LIN {X 0,Y 608.078,Z 640.045,A -85,B 0,C 180,E1 25976.717,E2 25976.717} C_VEL
LIN {X 0,Y 611.182,Z 594.743,A -85,B 0,C 180,E1 25973.511,E2 25973.511} C_VEL
LIN {X 0,Y 614.526,Z 550.793,A -85,B 0,C 180,E1 25970.32,E2 25970.32} C_VEL
LIN {X 0,Y 606.763,Z 531.048,A -85,B 0,C 180,E1 25968.076,E2 25968.076} C_VEL
LIN {X 0,Y 599.121,Z 513.107,A -85,B 0,C 180,E1 25965.86,E2 25965.86} C_VEL
LIN {X 0,Y 593.255,Z 499.729,A -85,B 0,C 180,E1 25964.077,E2 25964.077} C_VEL
LIN {X 0,Y 593.169,Z 499.296,A -85,B 0,C 180,E1 25963.406,E2 25963.406} C_VEL
LIN {X 0,Y 593.199,Z 499.34,A -85,B 0,C 180,E1 25960.21,E2 25960.21} C_VEL
LIN {X 0,Y 593.16,Z 499.3,A -85,B 0,C 180,E1 25956.966,E2 25956.966} C_VEL
LIN {X 0,Y 593.195,Z 499.329,A -85,B 0,C 180,E1 25953.797,E2 25953.797} C_VEL
LIN {X 0,Y 593.163,Z 499.335,A -85,B 0,C 180,E1 25950.603,E2 25950.603} C_VEL
LIN {X 0,Y 593.197,Z 499.328,A -85,B 0,C 180,E1 25947.398,E2 25947.398} C_VEL
LIN {X 0,Y 593.171,Z 499.341,A -85,B 0,C 180,E1 25944.181,E2 25944.181} C_VEL
LIN {X 0,Y 593.176,Z 499.338,A -85,B 0,C 180,E1 25940.835,E2 25940.835} C_VEL
LIN {X 0,Y 593.193,Z 499.334,A -85,B 0,C 180,E1 25937.663,E2 25937.663} C_VEL
LIN {X 0,Y 593.16,Z 499.324,A -85,B 0,C 180,E1 25934.447,E2 25934.447} C_VEL
LIN {X 0,Y 593.196,Z 499.326,A -85,B 0,C 180,E1 25931.276,E2 25931.276} C_VEL
LIN {X 0,Y 593.156,Z 499.342,A -85,B 0,C 180,E1 25928.043,E2 25928.043} C_VEL
LIN {X 0,Y 593.195,Z 499.331,A -85,B 0,C 180,E1 25924.835,E2 25924.835} C_VEL
LIN {X 0,Y 593.153,Z 499.332,A -85,B 0,C 180,E1 25921.739,E2 25921.739} C_VEL
LIN {X 0,Y 593.197,Z 499.336,A -85,B 0,C 180,E1 25918.551,E2 25918.551} C_VEL
LIN {X 0,Y 593.16,Z 499.332,A -85,B 0,C 180,E1 25915.359,E2 25915.359} C_VEL
LIN {X 0,Y 593.171,Z 499.319,A -85,B 0,C 180,E1 25912.055,E2 25912.055} C_VEL
LIN {X 0,Y 593.18,Z 499.34,A -85,B 0,C 180,E1 25908.921,E2 25908.921} C_VEL
LIN {X 0,Y 593.156,Z 499.34,A -85,B 0,C 180,E1 25905.653,E2 25905.653} C_VEL
LIN {X 0,Y 593.194,Z 499.326,A -85,B 0,C 180,E1 25902.54,E2 25902.54} C_VEL
LIN {X 0,Y 593.149,Z 499.33,A -85,B 0,C 180,E1 25899.317,E2 25899.317} C_VEL
LIN {X 0,Y 593.201,Z 499.331,A -85,B 0,C 180,E1 25896.24,E2 25896.24} C_VEL
LIN {X 0,Y 593.148,Z 499.344,A -85,B 0,C 180,E1 25893.034,E2 25893.034} C_VEL
LIN {X 0,Y 593.204,Z 499.341,A -85,B 0,C 180,E1 25889.959,E2 25889.959} C_VEL
LIN {X 0,Y 593.14,Z 499.291,A -85,B 0,C 180,E1 25886.779,E2 25886.779} C_VEL
LIN {X 0,Y 593.196,Z 499.341,A -85,B 0,C 180,E1 25883.606,E2 25883.606} C_VEL
LIN {X 0,Y 593.14,Z 499.296,A -85,B 0,C 180,E1 25880.538,E2 25880.538} C_VEL
LIN {X 0,Y 593.188,Z 499.306,A -85,B 0,C 180,E1 25877.342,E2 25877.342} C_VEL
LIN {X 0,Y 593.176,Z 499.54,A -85,B 0,C 180,E1 25876.313,E2 25876.313} C_VEL
LIN {X 0,Y 594.452,Z 502.746,A -85,B 0,C 180,E1 25875.864,E2 25875.864} C_VEL
LIN {X 0,Y 602.44,Z 520.278,A -85,B 0,C 180,E1 25873.643,E2 25873.643} C_VEL
LIN {X 0,Y 609.643,Z 537.266,A -85,B 0,C 180,E1 25871.662,E2 25871.662} C_VEL
LIN {X 0,Y 610.94,Z 539.957,A -85,B 0,C 180,E1 25871.41,E2 25871.41} C_VEL
LIN {X 0,Y 619.493,Z 554.552,A -85,B 0,C 180,E1 25870.572,E2 25870.572} C_VEL
LIN {X 0,Y 620.819,Z 562.667,A -85,B 0,C 180,E1 25870.357,E2 25870.357} C_VEL
LIN {X 0,Y 615.586,Z 815.185,A -85,B 0,C 180,E1 25866.946,E2 25866.946} C_VEL
LIN {X 0,Y 613.51,Z 921.471,A -85,B 0,C 180,E1 25865.506,E2 25865.506} C_VEL
LIN {X 0,Y 612.502,Z 946.347,A -85,B 0,C 180,E1 25865.008,E2 25865.008} C_VEL
LIN {X 0,Y 611.446,Z 967.057,A -85,B 0,C 180,E1 25864.465,E2 25864.465} C_VEL
LIN {X 0,Y 609.921,Z 992.831,A -85,B 0,C 180,E1 25863.612,E2 25863.612} C_VEL
LIN {X 0,Y 608.442,Z 1014.751,A -85,B 0,C 180,E1 25862.728,E2 25862.728} C_VEL
LIN {X 0,Y 606.737,Z 1038.002,A -85,B 0,C 180,E1 25861.604,E2 25861.604} C_VEL
LIN {X 0,Y 605.201,Z 1057.039,A -85,B 0,C 180,E1 25860.532,E2 25860.532} C_VEL
LIN {X 0,Y 603.232,Z 1079.697,A -85,B 0,C 180,E1 25859.055,E2 25859.055} C_VEL
LIN {X 0,Y 601.654,Z 1097.29,A -85,B 0,C 180,E1 25857.731,E2 25857.731} C_VEL
LIN {X 0,Y 599.985,Z 1115.676,A -85,B 0,C 180,E1 25856.154,E2 25856.154} C_VEL
LIN {X 0,Y 598.433,Z 1131.856,A -85,B 0,C 180,E1 25854.555,E2 25854.555} C_VEL
LIN {X 0,Y 596.98,Z 1147.996,A -85,B 0,C 180,E1 25852.761,E2 25852.761} C_VEL
LIN {X 0,Y 595.66,Z 1162.851,A -85,B 0,C 180,E1 25850.846,E2 25850.846} C_VEL
LIN {X 0,Y 594.748,Z 1173.87,A -85,B 0,C 180,E1 25849.239,E2 25849.239} C_VEL
LIN {X 0,Y 593.77,Z 1186.22,A -85,B 0,C 180,E1 25847.139,E2 25847.139} C_VEL
LIN {X 0,Y 593.053,Z 1196.639,A -85,B 0,C 180,E1 25845.048,E2 25845.048} C_VEL
LIN {X 0,Y 592.568,Z 1205.584,A -85,B 0,C 180,E1 25842.968,E2 25842.968} C_VEL
LIN {X 0,Y 592.211,Z 1213.908,A -85,B 0,C 180,E1 25840.605,E2 25840.605} C_VEL
LIN {X 0,Y 592.044,Z 1219.746,A -85,B 0,C 180,E1 25838.547,E2 25838.547} C_VEL
LIN {X 0,Y 591.951,Z 1225.015,A -85,B 0,C 180,E1 25836.109,E2 25836.109} C_VEL
LIN {X 0,Y 591.917,Z 1228.122,A -85,B 0,C 180,E1 25833.971,E2 25833.971} C_VEL
LIN {X 0,Y 591.899,Z 1230.037,A -85,B 0,C 180,E1 25831.742,E2 25831.742} C_VEL
LIN {X 0,Y 591.884,Z 1230.371,A -85,B 0,C 180,E1 25829.419,E2 25829.419} C_VEL
LIN {X 0,Y 591.892,Z 1229.426,A -85,B 0,C 180,E1 25827.386,E2 25827.386} C_VEL
LIN {X 0,Y 591.906,Z 1226.929,A -85,B 0,C 180,E1 25825.058,E2 25825.058} C_VEL
LIN {X 0,Y 591.973,Z 1223.102,A -85,B 0,C 180,E1 25822.917,E2 25822.917} C_VEL
LIN {X 0,Y 592.071,Z 1218.22,A -85,B 0,C 180,E1 25820.866,E2 25820.866} C_VEL
LIN {X 0,Y 592.321,Z 1210.66,A -85,B 0,C 180,E1 25818.412,E2 25818.412} C_VEL
LIN {X 0,Y 592.677,Z 1203.153,A -85,B 0,C 180,E1 25816.438,E2 25816.438} C_VEL
LIN {X 0,Y 593.283,Z 1193.273,A -85,B 0,C 180,E1 25814.226,E2 25814.226} C_VEL
LIN {X 0,Y 594.113,Z 1181.687,A -85,B 0,C 180,E1 25812.063,E2 25812.063} C_VEL
LIN {X 0,Y 595.01,Z 1170.617,A -85,B 0,C 180,E1 25810.259,E2 25810.259} C_VEL
LIN {X 0,Y 596.311,Z 1155.263,A -85,B 0,C 180,E1 25808.146,E2 25808.146} C_VEL
LIN {X 0,Y 597.61,Z 1140.965,A -85,B 0,C 180,E1 25806.43,E2 25806.43} C_VEL
LIN {X 0,Y 599.308,Z 1122.566,A -85,B 0,C 180,E1 25804.504,E2 25804.504} C_VEL
LIN {X 0,Y 600.868,Z 1105.911,A -85,B 0,C 180,E1 25802.982,E2 25802.982} C_VEL
LIN {X 0,Y 602.8,Z 1084.729,A -85,B 0,C 180,E1 25801.308,E2 25801.308} C_VEL
LIN {X 0,Y 604.418,Z 1066.075,A -85,B 0,C 180,E1 25800.028,E2 25800.028} C_VEL
LIN {X 0,Y 606.349,Z 1042.88,A -85,B 0,C 180,E1 25798.656,E2 25798.656} C_VEL
LIN {X 0,Y 607.897,Z 1022.873,A -85,B 0,C 180,E1 25797.644,E2 25797.644} C_VEL
LIN {X 0,Y 609.578,Z 998.087,A -85,B 0,C 180,E1 25796.586,E2 25796.586} C_VEL
LIN {X 0,Y 610.944,Z 975.646,A -85,B 0,C 180,E1 25795.794,E2 25795.794} C_VEL
LIN {X 0,Y 612.299,Z 950.422,A -85,B 0,C 180,E1 25795.088,E2 25795.088} C_VEL
LIN {X 0,Y 613.253,Z 928.821,A -85,B 0,C 180,E1 25794.626,E2 25794.626} C_VEL
LIN {X 0,Y 614.11,Z 895.917,A -85,B 0,C 180,E1 25794.131,E2 25794.131} C_VEL
LIN {X 0,Y 618.886,Z 652.893,A -85,B 0,C 180,E1 25790.86,E2 25790.86} C_VEL
LIN {X 0,Y 620.673,Z 560.775,A -85,B 0,C 180,E1 25789.605,E2 25789.605} C_VEL
LIN {X 0,Y 619.085,Z 553.518,A -85,B 0,C 180,E1 25789.385,E2 25789.385} C_VEL
LIN {X 0,Y 610.437,Z 539.117,A -85,B 0,C 180,E1 25788.537,E2 25788.537} C_VEL
LIN {X 0,Y 603.016,Z 521.573,A -85,B 0,C 180,E1 25786.519,E2 25786.519} C_VEL
LIN {X 0,Y 594.856,Z 503.322,A -85,B 0,C 180,E1 25784.233,E2 25784.233} C_VEL
LIN {X 0,Y 593.189,Z 499.611,A -85,B 0,C 180,E1 25783.718,E2 25783.718} C_VEL
LIN {X 0,Y 593.195,Z 499.309,A -85,B 0,C 180,E1 25782.526,E2 25782.526} C_VEL
LIN {X 0,Y 593.141,Z 499.295,A -85,B 0,C 180,E1 25779.46,E2 25779.46} C_VEL
LIN {X 0,Y 593.2,Z 499.341,A -85,B 0,C 180,E1 25776.324,E2 25776.324} C_VEL
LIN {X 0,Y 593.142,Z 499.291,A -85,B 0,C 180,E1 25773.106,E2 25773.106} C_VEL
LIN {X 0,Y 593.203,Z 499.342,A -85,B 0,C 180,E1 25769.929,E2 25769.929} C_VEL
LIN {X 0,Y 593.152,Z 499.343,A -85,B 0,C 180,E1 25766.858,E2 25766.858} C_VEL
LIN {X 0,Y 593.199,Z 499.333,A -85,B 0,C 180,E1 25763.651,E2 25763.651} C_VEL
LIN {X 0,Y 593.156,Z 499.331,A -85,B 0,C 180,E1 25760.526,E2 25760.526} C_VEL
LIN {X 0,Y 593.18,Z 499.327,A -85,B 0,C 180,E1 25757.258,E2 25757.258} C_VEL
LIN {X 0,Y 593.171,Z 499.339,A -85,B 0,C 180,E1 25754.148,E2 25754.148} C_VEL
LIN {X 0,Y 593.163,Z 499.344,A -85,B 0,C 180,E1 25750.784,E2 25750.784} C_VEL
LIN {X 0,Y 593.198,Z 499.317,A -85,B 0,C 180,E1 25747.652,E2 25747.652} C_VEL
LIN {X 0,Y 593.157,Z 499.329,A -85,B 0,C 180,E1 25744.447,E2 25744.447} C_VEL
LIN {X 0,Y 593.197,Z 499.337,A -85,B 0,C 180,E1 25741.256,E2 25741.256} C_VEL
LIN {X 0,Y 593.157,Z 499.334,A -85,B 0,C 180,E1 25738.068,E2 25738.068} C_VEL
LIN {X 0,Y 593.195,Z 499.327,A -85,B 0,C 180,E1 25734.875,E2 25734.875} C_VEL
LIN {X 0,Y 593.166,Z 499.339,A -85,B 0,C 180,E1 25731.675,E2 25731.675} C_VEL
LIN {X 0,Y 593.183,Z 499.335,A -85,B 0,C 180,E1 25728.328,E2 25728.328} C_VEL
LIN {X 0,Y 593.199,Z 499.319,A -85,B 0,C 180,E1 25725.055,E2 25725.055} C_VEL
LIN {X 0,Y 593.166,Z 499.33,A -85,B 0,C 180,E1 25721.829,E2 25721.829} C_VEL
LIN {X 0,Y 593.196,Z 499.339,A -85,B 0,C 180,E1 25718.648,E2 25718.648} C_VEL
LIN {X 0,Y 593.166,Z 499.343,A -85,B 0,C 180,E1 25715.501,E2 25715.501} C_VEL
LIN {X 0,Y 593.194,Z 499.331,A -85,B 0,C 180,E1 25712.275,E2 25712.275} C_VEL
LIN {X 0,Y 593.169,Z 499.337,A -85,B 0,C 180,E1 25709.09,E2 25709.09} C_VEL
LIN {X 0,Y 593.194,Z 499.332,A -85,B 0,C 180,E1 25705.853,E2 25705.853} C_VEL
LIN {X 0,Y 593.178,Z 499.293,A -85,B 0,C 180,E1 25702.639,E2 25702.639} C_VEL
LIN {X 0,Y 593.179,Z 499.342,A -85,B 0,C 180,E1 25699.281,E2 25699.281} C_VEL
LIN {X 0,Y 593.198,Z 499.367,A -85,B 0,C 180,E1 25696.015,E2 25696.015} C_VEL
LIN {X 0,Y 593.297,Z 499.956,A -85,B 0,C 180,E1 25695.79,E2 25695.79} C_VEL
LIN {X 0,Y 601.72,Z 518.947,A -85,B 0,C 180,E1 25693.295,E2 25693.295} C_VEL
LIN {X 0,Y 610.485,Z 540.277,A -85,B 0,C 180,E1 25690.754,E2 25690.754} C_VEL
LIN {X 0,Y 614.495,Z 551.086,A -85,B 0,C 180,E1 25689.564,E2 25689.564} C_VEL
LIN {X 0,Y 611.039,Z 596.556,A -85,B 0,C 180,E1 25686.266,E2 25686.266} C_VEL
LIN {X 0,Y 608.667,Z 630.364,A -85,B 0,C 180,E1 25683.868,E2 25683.868} C_VEL
LIN {X 0,Y 607.998,Z 636.114,A -85,B 0,C 180,E1 25683.565,E2 25683.565} C_VEL
LIN {X 0,Y 606.57,Z 644.568,A -85,B 0,C 180,E1 25683.334,E2 25683.334} C_VEL
LIN {X 0,Y 605.188,Z 656.769,A -85,B 0,C 180,E1 25683.155,E2 25683.155} C_VEL
LIN {X 0,Y 605.693,Z 664.458,A -85,B 0,C 180,E1 25683.005,E2 25683.005} C_VEL
LIN {X 0,Y 608.402,Z 681.191,A -85,B 0,C 180,E1 25682.592,E2 25682.592} C_VEL
LIN {X 0,Y 604.985,Z 954.452,A -85,B 0,C 180,E1 25679.305,E2 25679.305} C_VEL
LIN {X 0,Y 604.101,Z 976.225,A -85,B 0,C 180,E1 25678.892,E2 25678.892} C_VEL
LIN {X 0,Y 602.959,Z 997.031,A -85,B 0,C 180,E1 25678.338,E2 25678.338} C_VEL
LIN {X 0,Y 601.467,Z 1017.095,A -85,B 0,C 180,E1 25677.632,E2 25677.632} C_VEL
LIN {X 0,Y 599.717,Z 1037.712,A -85,B 0,C 180,E1 25676.726,E2 25676.726} C_VEL
LIN {X 0,Y 597.899,Z 1056.39,A -85,B 0,C 180,E1 25675.73,E2 25675.73} C_VEL
LIN {X 0,Y 595.886,Z 1074.87,A -85,B 0,C 180,E1 25674.543,E2 25674.543} C_VEL
LIN {X 0,Y 593.817,Z 1093.059,A -85,B 0,C 180,E1 25673.164,E2 25673.164} C_VEL
LIN {X 0,Y 591.871,Z 1109.557,A -85,B 0,C 180,E1 25671.696,E2 25671.696} C_VEL
LIN {X 0,Y 590.071,Z 1124.599,A -85,B 0,C 180,E1 25670.119,E2 25670.119} C_VEL
LIN {X 0,Y 588.473,Z 1138.59,A -85,B 0,C 180,E1 25668.423,E2 25668.423} C_VEL
LIN {X 0,Y 587.093,Z 1151.213,A -85,B 0,C 180,E1 25666.625,E2 25666.625} C_VEL
LIN {X 0,Y 585.924,Z 1163.106,A -85,B 0,C 180,E1 25664.625,E2 25664.625} C_VEL
LIN {X 0,Y 585.071,Z 1173.557,A -85,B 0,C 180,E1 25662.535,E2 25662.535} C_VEL
LIN {X 0,Y 584.502,Z 1182.555,A -85,B 0,C 180,E1 25660.347,E2 25660.347} C_VEL
LIN {X 0,Y 584.169,Z 1189.59,A -85,B 0,C 180,E1 25658.167,E2 25658.167} C_VEL
LIN {X 0,Y 583.993,Z 1194.928,A -85,B 0,C 180,E1 25655.995,E2 25655.995} C_VEL
LIN {X 0,Y 583.94,Z 1198.661,A -85,B 0,C 180,E1 25653.829,E2 25653.829} C_VEL
LIN {X 0,Y 583.918,Z 1200.67,A -85,B 0,C 180,E1 25651.668,E2 25651.668} C_VEL
LIN {X 0,Y 583.911,Z 1201.109,A -85,B 0,C 180,E1 25649.411,E2 25649.411} C_VEL
LIN {X 0,Y 583.927,Z 1199.973,A -85,B 0,C 180,E1 25647.252,E2 25647.252} C_VEL
LIN {X 0,Y 583.953,Z 1197.131,A -85,B 0,C 180,E1 25645.089,E2 25645.089} C_VEL
LIN {X 0,Y 584.053,Z 1192.685,A -85,B 0,C 180,E1 25642.92,E2 25642.92} C_VEL
LIN {X 0,Y 584.301,Z 1186.601,A -85,B 0,C 180,E1 25640.744,E2 25640.744} C_VEL
LIN {X 0,Y 584.701,Z 1179.023,A -85,B 0,C 180,E1 25638.659,E2 25638.659} C_VEL
LIN {X 0,Y 585.363,Z 1169.714,A -85,B 0,C 180,E1 25636.567,E2 25636.567} C_VEL
LIN {X 0,Y 586.305,Z 1159.134,A -85,B 0,C 180,E1 25634.572,E2 25634.572} C_VEL
LIN {X 0,Y 587.525,Z 1147.139,A -85,B 0,C 180,E1 25632.674,E2 25632.674} C_VEL
LIN {X 0,Y 589.006,Z 1133.769,A -85,B 0,C 180,E1 25630.875,E2 25630.875} C_VEL
LIN {X 0,Y 590.734,Z 1119.091,A -85,B 0,C 180,E1 25629.18,E2 25629.18} C_VEL
LIN {X 0,Y 592.539,Z 1103.888,A -85,B 0,C 180,E1 25627.687,E2 25627.687} C_VEL
LIN {X 0,Y 594.603,Z 1086.209,A -85,B 0,C 180,E1 25626.198,E2 25626.198} C_VEL
LIN {X 0,Y 596.657,Z 1068.291,A -85,B 0,C 180,E1 25624.915,E2 25624.915} C_VEL
LIN {X 0,Y 598.575,Z 1049.526,A -85,B 0,C 180,E1 25623.794,E2 25623.794} C_VEL
LIN {X 0,Y 600.524,Z 1028.723,A -85,B 0,C 180,E1 25622.764,E2 25622.764} C_VEL
LIN {X 0,Y 602.141,Z 1009.074,A -85,B 0,C 180,E1 25621.971,E2 25621.971} C_VEL
LIN {X 0,Y 603.476,Z 987.858,A -85,B 0,C 180,E1 25621.307,E2 25621.307} C_VEL
LIN {X 0,Y 604.607,Z 965.172,A -85,B 0,C 180,E1 25620.787,E2 25620.787} C_VEL
LIN {X 0,Y 605.264,Z 943.024,A -85,B 0,C 180,E1 25620.449,E2 25620.449} C_VEL
LIN {X 0,Y 608.386,Z 679.678,A -85,B 0,C 180,E1 25617.291,E2 25617.291} C_VEL
LIN {X 0,Y 601.204,Z 639.323,A -85,B 0,C 180,E1 25616.223,E2 25616.223} C_VEL
LIN {X 0,Y 604.486,Z 594.03,A -85,B 0,C 180,E1 25612.981,E2 25612.981} C_VEL
LIN {X 0,Y 607.7,Z 554.273,A -85,B 0,C 180,E1 25610.063,E2 25610.063} C_VEL
LIN {X 0,Y 599.505,Z 533.257,A -85,B 0,C 180,E1 25607.635,E2 25607.635} C_VEL
LIN {X 0,Y 591.378,Z 514.462,A -85,B 0,C 180,E1 25605.246,E2 25605.246} C_VEL
LIN {X 0,Y 586.57,Z 503.804,A -85,B 0,C 180,E1 25603.796,E2 25603.796} C_VEL
LIN {X 0,Y 585.256,Z 500.501,A -85,B 0,C 180,E1 25603.299,E2 25603.299} C_VEL
LIN {X 0,Y 585.26,Z 500.329,A -85,B 0,C 180,E1 25600.213,E2 25600.213} C_VEL
LIN {X 0,Y 585.221,Z 500.287,A -85,B 0,C 180,E1 25596.972,E2 25596.972} C_VEL
LIN {X 0,Y 585.256,Z 500.317,A -85,B 0,C 180,E1 25593.846,E2 25593.846} C_VEL
LIN {X 0,Y 585.224,Z 500.323,A -85,B 0,C 180,E1 25590.607,E2 25590.607} C_VEL
LIN {X 0,Y 585.257,Z 500.316,A -85,B 0,C 180,E1 25587.331,E2 25587.331} C_VEL
LIN {X 0,Y 585.237,Z 500.326,A -85,B 0,C 180,E1 25584.101,E2 25584.101} C_VEL
LIN {X 0,Y 585.23,Z 500.328,A -85,B 0,C 180,E1 25580.712,E2 25580.712} C_VEL
LIN {X 0,Y 585.258,Z 500.326,A -85,B 0,C 180,E1 25577.499,E2 25577.499} C_VEL
LIN {X 0,Y 585.217,Z 500.314,A -85,B 0,C 180,E1 25574.243,E2 25574.243} C_VEL
LIN {X 0,Y 585.256,Z 500.31,A -85,B 0,C 180,E1 25571.032,E2 25571.032} C_VEL
LIN {X 0,Y 585.22,Z 500.332,A -85,B 0,C 180,E1 25567.856,E2 25567.856} C_VEL
LIN {X 0,Y 585.251,Z 500.325,A -85,B 0,C 180,E1 25564.606,E2 25564.606} C_VEL
LIN {X 0,Y 585.226,Z 500.316,A -85,B 0,C 180,E1 25561.469,E2 25561.469} C_VEL
LIN {X 0,Y 585.227,Z 500.327,A -85,B 0,C 180,E1 25558.129,E2 25558.129} C_VEL
LIN {X 0,Y 585.255,Z 500.325,A -85,B 0,C 180,E1 25554.903,E2 25554.903} C_VEL
LIN {X 0,Y 585.213,Z 500.31,A -85,B 0,C 180,E1 25551.748,E2 25551.748} C_VEL
LIN {X 0,Y 585.258,Z 500.318,A -85,B 0,C 180,E1 25548.569,E2 25548.569} C_VEL
LIN {X 0,Y 585.209,Z 500.331,A -85,B 0,C 180,E1 25545.352,E2 25545.352} C_VEL
LIN {X 0,Y 585.259,Z 500.319,A -85,B 0,C 180,E1 25542.193,E2 25542.193} C_VEL
LIN {X 0,Y 585.211,Z 500.317,A -85,B 0,C 180,E1 25539.078,E2 25539.078} C_VEL
LIN {X 0,Y 585.257,Z 500.314,A -85,B 0,C 180,E1 25535.9,E2 25535.9} C_VEL
LIN {X 0,Y 585.216,Z 500.333,A -85,B 0,C 180,E1 25532.748,E2 25532.748} C_VEL
LIN {X 0,Y 585.231,Z 500.328,A -85,B 0,C 180,E1 25529.393,E2 25529.393} C_VEL
LIN {X 0,Y 585.228,Z 500.275,A -85,B 0,C 180,E1 25526.27,E2 25526.27} C_VEL
LIN {X 0,Y 585.215,Z 500.326,A -85,B 0,C 180,E1 25523.028,E2 25523.028} C_VEL
LIN {X 0,Y 585.249,Z 500.287,A -85,B 0,C 180,E1 25519.902,E2 25519.902} C_VEL
LIN {X 0,Y 585.256,Z 500.538,A -85,B 0,C 180,E1 25517.032,E2 25517.032} C_VEL
LIN {X 0,Y 586.504,Z 503.773,A -85,B 0,C 180,E1 25516.571,E2 25516.571} C_VEL
LIN {X 0,Y 591.053,Z 513.493,A -85,B 0,C 180,E1 25515.271,E2 25515.271} C_VEL
LIN {X 0,Y 599.255,Z 531.934,A -85,B 0,C 180,E1 25512.974,E2 25512.974} C_VEL
LIN {X 0,Y 602.865,Z 540.477,A -85,B 0,C 180,E1 25512.009,E2 25512.009} C_VEL
LIN {X 0,Y 613.481,Z 558.247,A -85,B 0,C 180,E1 25510.942,E2 25510.942} C_VEL
LIN {X 0,Y 614.388,Z 564.377,A -85,B 0,C 180,E1 25510.783,E2 25510.783} C_VEL
LIN {X 0,Y 608.882,Z 815.259,A -85,B 0,C 180,E1 25507.356,E2 25507.356} C_VEL
LIN {X 0,Y 606.647,Z 921.35,A -85,B 0,C 180,E1 25505.897,E2 25505.897} C_VEL
LIN {X 0,Y 605.592,Z 946.105,A -85,B 0,C 180,E1 25505.396,E2 25505.396} C_VEL
LIN {X 0,Y 604.471,Z 966.709,A -85,B 0,C 180,E1 25504.849,E2 25504.849} C_VEL
LIN {X 0,Y 602.89,Z 991.718,A -85,B 0,C 180,E1 25504.01,E2 25504.01} C_VEL
LIN {X 0,Y 601.315,Z 1013.033,A -85,B 0,C 180,E1 25503.136,E2 25503.136} C_VEL
LIN {X 0,Y 599.374,Z 1037.838,A -85,B 0,C 180,E1 25501.925,E2 25501.925} C_VEL
LIN {X 0,Y 597.77,Z 1056.876,A -85,B 0,C 180,E1 25500.842,E2 25500.842} C_VEL
LIN {X 0,Y 595.71,Z 1079.538,A -85,B 0,C 180,E1 25499.347,E2 25499.347} C_VEL
LIN {X 0,Y 594.056,Z 1097.142,A -85,B 0,C 180,E1 25498.007,E2 25498.007} C_VEL
LIN {X 0,Y 592.271,Z 1116.184,A -85,B 0,C 180,E1 25496.359,E2 25496.359} C_VEL
LIN {X 0,Y 590.707,Z 1132.035,A -85,B 0,C 180,E1 25494.781,E2 25494.781} C_VEL
LIN {X 0,Y 589.192,Z 1148.078,A -85,B 0,C 180,E1 25492.974,E2 25492.974} C_VEL
LIN {X 0,Y 587.812,Z 1162.906,A -85,B 0,C 180,E1 25491.033,E2 25491.033} C_VEL
LIN {X 0,Y 586.788,Z 1174.87,A -85,B 0,C 180,E1 25489.261,E2 25489.261} C_VEL
LIN {X 0,Y 585.746,Z 1188.213,A -85,B 0,C 180,E1 25486.971,E2 25486.971} C_VEL
LIN {X 0,Y 585.12,Z 1197.097,A -85,B 0,C 180,E1 25485.156,E2 25485.156} C_VEL
LIN {X 0,Y 584.563,Z 1206.776,A -85,B 0,C 180,E1 25482.847,E2 25482.847} C_VEL
LIN {X 0,Y 584.21,Z 1214.514,A -85,B 0,C 180,E1 25480.552,E2 25480.552} C_VEL
LIN {X 0,Y 584.047,Z 1220.509,A -85,B 0,C 180,E1 25478.367,E2 25478.367} C_VEL
LIN {X 0,Y 583.947,Z 1225.334,A -85,B 0,C 180,E1 25475.995,E2 25475.995} C_VEL
LIN {X 0,Y 583.916,Z 1228.235,A -85,B 0,C 180,E1 25473.927,E2 25473.927} C_VEL
LIN {X 0,Y 583.897,Z 1230.144,A -85,B 0,C 180,E1 25471.57,E2 25471.57} C_VEL
LIN {X 0,Y 583.885,Z 1230.348,A -85,B 0,C 180,E1 25469.313,E2 25469.313} C_VEL
LIN {X 0,Y 583.891,Z 1229.426,A -85,B 0,C 180,E1 25467.35,E2 25467.35} C_VEL
LIN {X 0,Y 583.905,Z 1226.929,A -85,B 0,C 180,E1 25464.99,E2 25464.99} C_VEL
LIN {X 0,Y 583.971,Z 1223.102,A -85,B 0,C 180,E1 25462.82,E2 25462.82} C_VEL
LIN {X 0,Y 584.091,Z 1218.22,A -85,B 0,C 180,E1 25460.74,E2 25460.74} C_VEL
LIN {X 0,Y 584.364,Z 1210.66,A -85,B 0,C 180,E1 25458.252,E2 25458.252} C_VEL
LIN {X 0,Y 584.746,Z 1203.072,A -85,B 0,C 180,E1 25456.23,E2 25456.23} C_VEL
LIN {X 0,Y 585.416,Z 1192.916,A -85,B 0,C 180,E1 25453.937,E2 25453.937} C_VEL
LIN {X 0,Y 586.215,Z 1181.999,A -85,B 0,C 180,E1 25451.915,E2 25451.915} C_VEL
LIN {X 0,Y 587.201,Z 1170.018,A -85,B 0,C 180,E1 25449.986,E2 25449.986} C_VEL
LIN {X 0,Y 588.494,Z 1155.34,A -85,B 0,C 180,E1 25447.946,E2 25447.946} C_VEL
LIN {X 0,Y 589.854,Z 1141.031,A -85,B 0,C 180,E1 25446.207,E2 25446.207} C_VEL
LIN {X 0,Y 591.607,Z 1122.737,A -85,B 0,C 180,E1 25444.269,E2 25444.269} C_VEL
LIN {X 0,Y 593.247,Z 1105.809,A -85,B 0,C 180,E1 25442.714,E2 25442.714} C_VEL
LIN {X 0,Y 595.263,Z 1084.514,A -85,B 0,C 180,E1 25441.014,E2 25441.014} C_VEL
LIN {X 0,Y 596.993,Z 1065.429,A -85,B 0,C 180,E1 25439.693,E2 25439.693} C_VEL
LIN {X 0,Y 598.985,Z 1042.62,A -85,B 0,C 180,E1 25438.333,E2 25438.333} C_VEL
LIN {X 0,Y 600.704,Z 1021.482,A -85,B 0,C 180,E1 25437.251,E2 25437.251} C_VEL
LIN {X 0,Y 602.446,Z 997.731,A -85,B 0,C 180,E1 25436.221,E2 25436.221} C_VEL
LIN {X 0,Y 603.859,Z 976.413,A -85,B 0,C 180,E1 25435.452,E2 25435.452} C_VEL
LIN {X 0,Y 605.34,Z 950.895,A -85,B 0,C 180,E1 25434.719,E2 25434.719} C_VEL
LIN {X 0,Y 606.335,Z 929.724,A -85,B 0,C 180,E1 25434.256,E2 25434.256} C_VEL
LIN {X 0,Y 607.218,Z 899.395,A -85,B 0,C 180,E1 25433.784,E2 25433.784} C_VEL
LIN {X 0,Y 612.363,Z 653.966,A -85,B 0,C 180,E1 25430.437,E2 25430.437} C_VEL
LIN {X 0,Y 614.25,Z 562.382,A -85,B 0,C 180,E1 25429.177,E2 25429.177} C_VEL
LIN {X 0,Y 613.083,Z 557.386,A -85,B 0,C 180,E1 25429.018,E2 25429.018} C_VEL
LIN {X 0,Y 602.567,Z 539.941,A -85,B 0,C 180,E1 25427.952,E2 25427.952} C_VEL
LIN {X 0,Y 594.327,Z 520.546,A -85,B 0,C 180,E1 25425.645,E2 25425.645} C_VEL
LIN {X 0,Y 587.957,Z 506.912,A -85,B 0,C 180,E1 25423.86,E2 25423.86} C_VEL
LIN {X 0,Y 585.275,Z 500.681,A -85,B 0,C 180,E1 25423.015,E2 25423.015} C_VEL
LIN {X 0,Y 585.259,Z 500.303,A -85,B 0,C 180,E1 25422.291,E2 25422.291} C_VEL
LIN {X 0,Y 585.201,Z 500.28,A -85,B 0,C 180,E1 25419.212,E2 25419.212} C_VEL
LIN {X 0,Y 585.253,Z 500.33,A -85,B 0,C 180,E1 25415.995,E2 25415.995} C_VEL
LIN {X 0,Y 585.215,Z 500.278,A -85,B 0,C 180,E1 25412.794,E2 25412.794} C_VEL
LIN {X 0,Y 585.227,Z 500.326,A -85,B 0,C 180,E1 25409.476,E2 25409.476} C_VEL
LIN {X 0,Y 585.242,Z 500.329,A -85,B 0,C 180,E1 25406.373,E2 25406.373} C_VEL
LIN {X 0,Y 585.219,Z 500.334,A -85,B 0,C 180,E1 25403.14,E2 25403.14} C_VEL
LIN {X 0,Y 585.257,Z 500.318,A -85,B 0,C 180,E1 25399.98,E2 25399.98} C_VEL
LIN {X 0,Y 585.214,Z 500.317,A -85,B 0,C 180,E1 25396.783,E2 25396.783} C_VEL
LIN {X 0,Y 585.262,Z 500.321,A -85,B 0,C 180,E1 25393.637,E2 25393.637} C_VEL
LIN {X 0,Y 585.216,Z 500.33,A -85,B 0,C 180,E1 25390.434,E2 25390.434} C_VEL
LIN {X 0,Y 585.261,Z 500.312,A -85,B 0,C 180,E1 25387.164,E2 25387.164} C_VEL
LIN {X 0,Y 585.223,Z 500.314,A -85,B 0,C 180,E1 25384.017,E2 25384.017} C_VEL
LIN {X 0,Y 585.243,Z 500.327,A -85,B 0,C 180,E1 25380.685,E2 25380.685} C_VEL
LIN {X 0,Y 585.25,Z 500.321,A -85,B 0,C 180,E1 25377.454,E2 25377.454} C_VEL
LIN {X 0,Y 585.224,Z 500.314,A -85,B 0,C 180,E1 25374.214,E2 25374.214} C_VEL
LIN {X 0,Y 585.259,Z 500.327,A -85,B 0,C 180,E1 25371.056,E2 25371.056} C_VEL
LIN {X 0,Y 585.223,Z 500.332,A -85,B 0,C 180,E1 25367.869,E2 25367.869} C_VEL
LIN {X 0,Y 585.255,Z 500.311,A -85,B 0,C 180,E1 25364.644,E2 25364.644} C_VEL
LIN {X 0,Y 585.225,Z 500.316,A -85,B 0,C 180,E1 25361.47,E2 25361.47} C_VEL
LIN {X 0,Y 585.258,Z 500.322,A -85,B 0,C 180,E1 25358.133,E2 25358.133} C_VEL
LIN {X 0,Y 585.253,Z 500.327,A -85,B 0,C 180,E1 25354.823,E2 25354.823} C_VEL
LIN {X 0,Y 585.232,Z 500.333,A -85,B 0,C 180,E1 25351.531,E2 25351.531} C_VEL
LIN {X 0,Y 585.258,Z 500.327,A -85,B 0,C 180,E1 25348.365,E2 25348.365} C_VEL
LIN {X 0,Y 585.232,Z 500.333,A -85,B 0,C 180,E1 25345.085,E2 25345.085} C_VEL
LIN {X 0,Y 585.249,Z 500.276,A -85,B 0,C 180,E1 25341.795,E2 25341.795} C_VEL
LIN {X 0,Y 585.237,Z 500.306,A -85,B 0,C 180,E1 25338.592,E2 25338.592} C_VEL
LIN {X 0,Y 585.274,Z 500.55,A -85,B 0,C 180,E1 25336.579,E2 25336.579} C_VEL
LIN {X 0,Y 588.491,Z 507.938,A -85,B 0,C 180,E1 25335.527,E2 25335.527} C_VEL
LIN {X 0,Y 595.828,Z 524.591,A -85,B 0,C 180,E1 25333.341,E2 25333.341} C_VEL
LIN {X 0,Y 604.237,Z 545.17,A -85,B 0,C 180,E1 25330.866,E2 25330.866} C_VEL
LIN {X 0,Y 607.676,Z 554.478,A -85,B 0,C 180,E1 25329.826,E2 25329.826} C_VEL
LIN {X 0,Y 604.049,Z 599.651,A -85,B 0,C 180,E1 25326.517,E2 25326.517} C_VEL
LIN {X 0,Y 601.247,Z 639.999,A -85,B 0,C 180,E1 25323.656,E2 25323.656} C_VEL
LIN {X 0,Y 605.693,Z 664.458,A -85,B 0,C 180,E1 25323.005,E2 25323.005} C_VEL
LIN {X 0,Y 606.078,Z 670.985,A -85,B 0,C 180,E1 25322.89,E2 25322.89} C_VEL
LIN {X 0,Y 604.74,Z 680.96,A -85,B 0,C 180,E1 25322.849,E2 25322.849} C_VEL
LIN {X 0,Y 601.98,Z 695.522,A -85,B 0,C 180,E1 25322.847,E2 25322.847} C_VEL
LIN {X 0,Y 601.669,Z 700.04,A -85,B 0,C 180,E1 25322.809,E2 25322.809} C_VEL
LIN {X 0,Y 598.289,Z 954.495,A -85,B 0,C 180,E1 25319.724,E2 25319.724} C_VEL
LIN {X 0,Y 597.355,Z 976.226,A -85,B 0,C 180,E1 25319.307,E2 25319.307} C_VEL
LIN {X 0,Y 596.146,Z 997.126,A -85,B 0,C 180,E1 25318.746,E2 25318.746} C_VEL
LIN {X 0,Y 594.579,Z 1017.307,A -85,B 0,C 180,E1 25318.03,E2 25318.03} C_VEL
LIN {X 0,Y 592.694,Z 1038.275,A -85,B 0,C 180,E1 25317.096,E2 25317.096} C_VEL
LIN {X 0,Y 590.729,Z 1057.529,A -85,B 0,C 180,E1 25316.054,E2 25316.054} C_VEL
LIN {X 0,Y 588.637,Z 1075.699,A -85,B 0,C 180,E1 25314.865,E2 25314.865} C_VEL
LIN {X 0,Y 586.366,Z 1094.513,A -85,B 0,C 180,E1 25313.41,E2 25313.41} C_VEL
LIN {X 0,Y 584.31,Z 1111.091,A -85,B 0,C 180,E1 25311.903,E2 25311.903} C_VEL
LIN {X 0,Y 582.412,Z 1126.124,A -85,B 0,C 180,E1 25310.291,E2 25310.291} C_VEL
LIN {X 0,Y 580.646,Z 1140.659,A -85,B 0,C 180,E1 25308.472,E2 25308.472} C_VEL
LIN {X 0,Y 579.238,Z 1153.148,A -85,B 0,C 180,E1 25306.651,E2 25306.651} C_VEL
LIN {X 0,Y 578.022,Z 1164.762,A -85,B 0,C 180,E1 25304.628,E2 25304.628} C_VEL
LIN {X 0,Y 577.125,Z 1174.932,A -85,B 0,C 180,E1 25302.507,E2 25302.507} C_VEL
LIN {X 0,Y 576.55,Z 1183.311,A -85,B 0,C 180,E1 25300.391,E2 25300.391} C_VEL
LIN {X 0,Y 576.195,Z 1190.227,A -85,B 0,C 180,E1 25298.181,E2 25298.181} C_VEL
LIN {X 0,Y 576.004,Z 1195.409,A -85,B 0,C 180,E1 25295.978,E2 25295.978} C_VEL
LIN {X 0,Y 575.943,Z 1199.001,A -85,B 0,C 180,E1 25293.783,E2 25293.783} C_VEL
LIN {X 0,Y 575.922,Z 1200.883,A -85,B 0,C 180,E1 25291.691,E2 25291.691} C_VEL
LIN {X 0,Y 575.914,Z 1201.314,A -85,B 0,C 180,E1 25289.403,E2 25289.403} C_VEL
LIN {X 0,Y 575.931,Z 1200.194,A -85,B 0,C 180,E1 25287.214,E2 25287.214} C_VEL
LIN {X 0,Y 575.959,Z 1197.529,A -85,B 0,C 180,E1 25285.12,E2 25285.12} C_VEL
LIN {X 0,Y 576.079,Z 1192.986,A -85,B 0,C 180,E1 25282.821,E2 25282.821} C_VEL
LIN {X 0,Y 576.352,Z 1186.984,A -85,B 0,C 180,E1 25280.615,E2 25280.615} C_VEL
LIN {X 0,Y 576.792,Z 1179.477,A -85,B 0,C 180,E1 25278.501,E2 25278.501} C_VEL
LIN {X 0,Y 577.521,Z 1170.273,A -85,B 0,C 180,E1 25276.382,E2 25276.382} C_VEL
LIN {X 0,Y 578.532,Z 1159.746,A -85,B 0,C 180,E1 25274.359,E2 25274.359} C_VEL
LIN {X 0,Y 579.827,Z 1147.718,A -85,B 0,C 180,E1 25272.436,E2 25272.436} C_VEL
LIN {X 0,Y 581.398,Z 1134.379,A -85,B 0,C 180,E1 25270.615,E2 25270.615} C_VEL
LIN {X 0,Y 583.225,Z 1119.749,A -85,B 0,C 180,E1 25268.899,E2 25268.899} C_VEL
LIN {X 0,Y 585.222,Z 1103.771,A -85,B 0,C 180,E1 25267.314,E2 25267.314} C_VEL
LIN {X 0,Y 587.344,Z 1086.557,A -85,B 0,C 180,E1 25265.851,E2 25265.851} C_VEL
LIN {X 0,Y 589.53,Z 1068.382,A -85,B 0,C 180,E1 25264.536,E2 25264.536} C_VEL
LIN {X 0,Y 591.574,Z 1049.368,A -85,B 0,C 180,E1 25263.391,E2 25263.391} C_VEL
LIN {X 0,Y 593.558,Z 1029.248,A -85,B 0,C 180,E1 25262.386,E2 25262.386} C_VEL
LIN {X 0,Y 595.289,Z 1009.133,A -85,B 0,C 180,E1 25261.564,E2 25261.564} C_VEL
LIN {X 0,Y 596.699,Z 987.926,A -85,B 0,C 180,E1 25260.895,E2 25260.895} C_VEL
LIN {X 0,Y 597.894,Z 965.132,A -85,B 0,C 180,E1 25260.368,E2 25260.368} C_VEL
LIN {X 0,Y 598.587,Z 943.016,A -85,B 0,C 180,E1 25260.027,E2 25260.027} C_VEL
LIN {X 0,Y 601.923,Z 681.148,A -85,B 0,C 180,E1 25256.859,E2 25256.859} C_VEL
LIN {X 0,Y 594.362,Z 638.132,A -85,B 0,C 180,E1 25255.691,E2 25255.691} C_VEL
LIN {X 0,Y 597.906,Z 592.557,A -85,B 0,C 180,E1 25252.383,E2 25252.383} C_VEL
LIN {X 0,Y 600.846,Z 557.613,A -85,B 0,C 180,E1 25249.785,E2 25249.785} C_VEL
LIN {X 0,Y 592.939,Z 537.286,A -85,B 0,C 180,E1 25247.399,E2 25247.399} C_VEL
LIN {X 0,Y 584.416,Z 517.303,A -85,B 0,C 180,E1 25244.822,E2 25244.822} C_VEL
LIN {X 0,Y 578.448,Z 504.541,A -85,B 0,C 180,E1 25243.016,E2 25243.016} C_VEL
LIN {X 0,Y 577.33,Z 501.463,A -85,B 0,C 180,E1 25242.537,E2 25242.537} C_VEL
LIN {X 0,Y 577.289,Z 501.285,A -85,B 0,C 180,E1 25239.213,E2 25239.213} C_VEL
LIN {X 0,Y 577.317,Z 501.298,A -85,B 0,C 180,E1 25235.954,E2 25235.954} C_VEL
LIN {X 0,Y 577.285,Z 501.313,A -85,B 0,C 180,E1 25232.675,E2 25232.675} C_VEL
LIN {X 0,Y 577.322,Z 501.311,A -85,B 0,C 180,E1 25229.409,E2 25229.409} C_VEL
LIN {X 0,Y 577.303,Z 501.306,A -85,B 0,C 180,E1 25226.1,E2 25226.1} C_VEL
LIN {X 0,Y 577.288,Z 501.301,A -85,B 0,C 180,E1 25222.721,E2 25222.721} C_VEL
LIN {X 0,Y 577.319,Z 501.3,A -85,B 0,C 180,E1 25219.528,E2 25219.528} C_VEL
LIN {X 0,Y 577.281,Z 501.32,A -85,B 0,C 180,E1 25216.296,E2 25216.296} C_VEL
LIN {X 0,Y 577.321,Z 501.318,A -85,B 0,C 180,E1 25213.114,E2 25213.114} C_VEL
LIN {X 0,Y 577.282,Z 501.301,A -85,B 0,C 180,E1 25209.874,E2 25209.874} C_VEL
LIN {X 0,Y 577.305,Z 501.304,A -85,B 0,C 180,E1 25206.564,E2 25206.564} C_VEL
LIN {X 0,Y 577.309,Z 501.321,A -85,B 0,C 180,E1 25203.277,E2 25203.277} C_VEL
LIN {X 0,Y 577.279,Z 501.312,A -85,B 0,C 180,E1 25200,E2 25200} C_VEL
LIN {X 0,Y 577.318,Z 501.298,A -85,B 0,C 180,E1 25196.823,E2 25196.823} C_VEL
LIN {X 0,Y 577.276,Z 501.32,A -85,B 0,C 180,E1 25193.635,E2 25193.635} C_VEL
LIN {X 0,Y 577.321,Z 501.315,A -85,B 0,C 180,E1 25190.429,E2 25190.429} C_VEL
LIN {X 0,Y 577.278,Z 501.302,A -85,B 0,C 180,E1 25187.191,E2 25187.191} C_VEL
LIN {X 0,Y 577.301,Z 501.306,A -85,B 0,C 180,E1 25183.911,E2 25183.911} C_VEL
LIN {X 0,Y 577.301,Z 501.32,A -85,B 0,C 180,E1 25180.682,E2 25180.682} C_VEL
LIN {X 0,Y 577.277,Z 501.319,A -85,B 0,C 180,E1 25177.386,E2 25177.386} C_VEL
LIN {X 0,Y 577.318,Z 501.308,A -85,B 0,C 180,E1 25174.232,E2 25174.232} C_VEL
LIN {X 0,Y 577.268,Z 501.312,A -85,B 0,C 180,E1 25170.988,E2 25170.988} C_VEL
LIN {X 0,Y 577.317,Z 501.272,A -85,B 0,C 180,E1 25167.876,E2 25167.876} C_VEL
LIN {X 0,Y 577.268,Z 501.306,A -85,B 0,C 180,E1 25164.653,E2 25164.653} C_VEL
LIN {X 0,Y 577.313,Z 501.263,A -85,B 0,C 180,E1 25161.427,E2 25161.427} C_VEL
LIN {X 0,Y 577.274,Z 501.318,A -85,B 0,C 180,E1 25158.288,E2 25158.288} C_VEL
LIN {X 0,Y 577.388,Z 501.747,A -85,B 0,C 180,E1 25157.733,E2 25157.733} C_VEL
LIN {X 0,Y 579.062,Z 505.428,A -85,B 0,C 180,E1 25157.197,E2 25157.197} C_VEL
LIN {X 0,Y 587.059,Z 523.033,A -85,B 0,C 180,E1 25154.838,E2 25154.838} C_VEL
LIN {X 0,Y 595.089,Z 541.406,A -85,B 0,C 180,E1 25152.595,E2 25152.595} C_VEL
LIN {X 0,Y 607.479,Z 561.87,A -85,B 0,C 180,E1 25151.321,E2 25151.321} C_VEL
LIN {X 0,Y 607.994,Z 566.125,A -85,B 0,C 180,E1 25151.218,E2 25151.218} C_VEL
LIN {X 0,Y 602.239,Z 814.354,A -85,B 0,C 180,E1 25147.79,E2 25147.79} C_VEL
LIN {X 0,Y 599.838,Z 921.394,A -85,B 0,C 180,E1 25146.299,E2 25146.299} C_VEL
LIN {X 0,Y 598.732,Z 946.148,A -85,B 0,C 180,E1 25145.792,E2 25145.792} C_VEL
LIN {X 0,Y 597.541,Z 966.898,A -85,B 0,C 180,E1 25145.234,E2 25145.234} C_VEL
LIN {X 0,Y 595.9,Z 991.402,A -85,B 0,C 180,E1 25144.402,E2 25144.402} C_VEL
LIN {X 0,Y 594.295,Z 1011.932,A -85,B 0,C 180,E1 25143.551,E2 25143.551} C_VEL
LIN {X 0,Y 592.333,Z 1035.151,A -85,B 0,C 180,E1 25142.413,E2 25142.413} C_VEL
LIN {X 0,Y 590.441,Z 1055.945,A -85,B 0,C 180,E1 25141.21,E2 25141.21} C_VEL
LIN {X 0,Y 588.309,Z 1078.453,A -85,B 0,C 180,E1 25139.715,E2 25139.715} C_VEL
LIN {X 0,Y 586.54,Z 1096.363,A -85,B 0,C 180,E1 25138.343,E2 25138.343} C_VEL
LIN {X 0,Y 584.666,Z 1115.521,A -85,B 0,C 180,E1 25136.674,E2 25136.674} C_VEL
LIN {X 0,Y 582.975,Z 1132.047,A -85,B 0,C 180,E1 25135.014,E2 25135.014} C_VEL
LIN {X 0,Y 581.41,Z 1148.144,A -85,B 0,C 180,E1 25133.192,E2 25133.192} C_VEL
LIN {X 0,Y 579.971,Z 1162.973,A -85,B 0,C 180,E1 25131.225,E2 25131.225} C_VEL
LIN {X 0,Y 578.867,Z 1175.33,A -85,B 0,C 180,E1 25129.368,E2 25129.368} C_VEL
LIN {X 0,Y 577.809,Z 1188.248,A -85,B 0,C 180,E1 25127.108,E2 25127.108} C_VEL
LIN {X 0,Y 577.139,Z 1197.779,A -85,B 0,C 180,E1 25125.165,E2 25125.165} C_VEL
LIN {X 0,Y 576.598,Z 1207.13,A -85,B 0,C 180,E1 25122.926,E2 25122.926} C_VEL
LIN {X 0,Y 576.243,Z 1214.513,A -85,B 0,C 180,E1 25120.7,E2 25120.7} C_VEL
LIN {X 0,Y 576.052,Z 1220.763,A -85,B 0,C 180,E1 25118.384,E2 25118.384} C_VEL
LIN {X 0,Y 575.947,Z 1225.494,A -85,B 0,C 180,E1 25115.979,E2 25115.979} C_VEL
LIN {X 0,Y 575.915,Z 1228.349,A -85,B 0,C 180,E1 25113.882,E2 25113.882} C_VEL
LIN {X 0,Y 575.901,Z 1230.189,A -85,B 0,C 180,E1 25111.393,E2 25111.393} C_VEL
LIN {X 0,Y 575.886,Z 1230.348,A -85,B 0,C 180,E1 25109.304,E2 25109.304} C_VEL
LIN {X 0,Y 575.889,Z 1229.425,A -85,B 0,C 180,E1 25107.313,E2 25107.313} C_VEL
LIN {X 0,Y 575.905,Z 1226.929,A -85,B 0,C 180,E1 25104.92,E2 25104.92} C_VEL
LIN {X 0,Y 575.97,Z 1223.102,A -85,B 0,C 180,E1 25102.72,E2 25102.72} C_VEL
LIN {X 0,Y 576.099,Z 1218.475,A -85,B 0,C 180,E1 25100.711,E2 25100.711} C_VEL
LIN {X 0,Y 576.39,Z 1211.013,A -85,B 0,C 180,E1 25098.188,E2 25098.188} C_VEL
LIN {X 0,Y 576.759,Z 1203.905,A -85,B 0,C 180,E1 25096.261,E2 25096.261} C_VEL
LIN {X 0,Y 577.335,Z 1194.962,A -85,B 0,C 180,E1 25094.223,E2 25094.223} C_VEL
LIN {X 0,Y 578.255,Z 1182.651,A -85,B 0,C 180,E1 25091.866,E2 25091.866} C_VEL
LIN {X 0,Y 579.202,Z 1171.391,A -85,B 0,C 180,E1 25090.013,E2 25090.013} C_VEL
LIN {X 0,Y 580.609,Z 1156.21,A -85,B 0,C 180,E1 25087.844,E2 25087.844} C_VEL
LIN {X 0,Y 581.916,Z 1142.816,A -85,B 0,C 180,E1 25086.185,E2 25086.185} C_VEL
LIN {X 0,Y 583.589,Z 1126.229,A -85,B 0,C 180,E1 25084.367,E2 25084.367} C_VEL
LIN {X 0,Y 585.385,Z 1108.032,A -85,B 0,C 180,E1 25082.648,E2 25082.648} C_VEL
LIN {X 0,Y 587.329,Z 1088.85,A -85,B 0,C 180,E1 25081.052,E2 25081.052} C_VEL
LIN {X 0,Y 589.279,Z 1068.095,A -85,B 0,C 180,E1 25079.57,E2 25079.57} C_VEL
LIN {X 0,Y 591.41,Z 1045.572,A -85,B 0,C 180,E1 25078.165,E2 25078.165} C_VEL
LIN {X 0,Y 593.217,Z 1025.165,A -85,B 0,C 180,E1 25077.077,E2 25077.077} C_VEL
LIN {X 0,Y 595.078,Z 1002.556,A -85,B 0,C 180,E1 25076.036,E2 25076.036} C_VEL
LIN {X 0,Y 596.722,Z 979.031,A -85,B 0,C 180,E1 25075.154,E2 25075.154} C_VEL
LIN {X 0,Y 598.259,Z 954.768,A -85,B 0,C 180,E1 25074.418,E2 25074.418} C_VEL
LIN {X 0,Y 599.403,Z 931.987,A -85,B 0,C 180,E1 25073.9,E2 25073.9} C_VEL
LIN {X 0,Y 600.281,Z 907.035,A -85,B 0,C 180,E1 25073.482,E2 25073.482} C_VEL
LIN {X 0,Y 605.767,Z 659.787,A -85,B 0,C 180,E1 25070.071,E2 25070.071} C_VEL
LIN {X 0,Y 607.863,Z 563.975,A -85,B 0,C 180,E1 25068.741,E2 25068.741} C_VEL
LIN {X 0,Y 607.025,Z 561.065,A -85,B 0,C 180,E1 25068.634,E2 25068.634} C_VEL
LIN {X 0,Y 594.764,Z 540.792,A -85,B 0,C 180,E1 25067.353,E2 25067.353} C_VEL
LIN {X 0,Y 586.222,Z 521.086,A -85,B 0,C 180,E1 25064.922,E2 25064.922} C_VEL
LIN {X 0,Y 580.272,Z 508.413,A -85,B 0,C 180,E1 25063.209,E2 25063.209} C_VEL
LIN {X 0,Y 577.347,Z 501.514,A -85,B 0,C 180,E1 25062.232,E2 25062.232} C_VEL
LIN {X 0,Y 577.262,Z 501.267,A -85,B 0,C 180,E1 25059.215,E2 25059.215} C_VEL
LIN {X 0,Y 577.312,Z 501.318,A -85,B 0,C 180,E1 25055.955,E2 25055.955} C_VEL
LIN {X 0,Y 577.274,Z 501.264,A -85,B 0,C 180,E1 25052.83,E2 25052.83} C_VEL
LIN {X 0,Y 577.288,Z 501.315,A -85,B 0,C 180,E1 25049.466,E2 25049.466} C_VEL
LIN {X 0,Y 577.308,Z 501.319,A -85,B 0,C 180,E1 25046.32,E2 25046.32} C_VEL
LIN {X 0,Y 577.278,Z 501.322,A -85,B 0,C 180,E1 25043.045,E2 25043.045} C_VEL
LIN {X 0,Y 577.321,Z 501.308,A -85,B 0,C 180,E1 25039.844,E2 25039.844} C_VEL
LIN {X 0,Y 577.275,Z 501.306,A -85,B 0,C 180,E1 25036.606,E2 25036.606} C_VEL
LIN {X 0,Y 577.319,Z 501.305,A -85,B 0,C 180,E1 25033.42,E2 25033.42} C_VEL
LIN {X 0,Y 577.286,Z 501.318,A -85,B 0,C 180,E1 25030.176,E2 25030.176} C_VEL
LIN {X 0,Y 577.291,Z 501.313,A -85,B 0,C 180,E1 25026.764,E2 25026.764} C_VEL
LIN {X 0,Y 577.311,Z 501.296,A -85,B 0,C 180,E1 25023.575,E2 25023.575} C_VEL
LIN {X 0,Y 577.281,Z 501.313,A -85,B 0,C 180,E1 25020.298,E2 25020.298} C_VEL
LIN {X 0,Y 577.32,Z 501.312,A -85,B 0,C 180,E1 25017.121,E2 25017.121} C_VEL
LIN {X 0,Y 577.281,Z 501.302,A -85,B 0,C 180,E1 25013.935,E2 25013.935} C_VEL
LIN {X 0,Y 577.317,Z 501.308,A -85,B 0,C 180,E1 25010.731,E2 25010.731} C_VEL
LIN {X 0,Y 577.294,Z 501.318,A -85,B 0,C 180,E1 25007.496,E2 25007.496} C_VEL
LIN {X 0,Y 577.301,Z 501.31,A -85,B 0,C 180,E1 25004.118,E2 25004.118} C_VEL
LIN {X 0,Y 577.316,Z 501.298,A -85,B 0,C 180,E1 25000.892,E2 25000.892} C_VEL
LIN {X 0,Y 577.287,Z 501.305,A -85,B 0,C 180,E1 24997.601,E2 24997.601} C_VEL
LIN {X 0,Y 577.316,Z 501.314,A -85,B 0,C 180,E1 24994.342,E2 24994.342} C_VEL
LIN {X 0,Y 577.294,Z 501.318,A -85,B 0,C 180,E1 24991.103,E2 24991.103} C_VEL
LIN {X 0,Y 577.314,Z 501.317,A -85,B 0,C 180,E1 24987.761,E2 24987.761} C_VEL
LIN {X 0,Y 577.318,Z 501.312,A -85,B 0,C 180,E1 24984.413,E2 24984.413} C_VEL
LIN {X 0,Y 577.288,Z 501.273,A -85,B 0,C 180,E1 24981.171,E2 24981.171} C_VEL
LIN {X 0,Y 577.311,Z 501.275,A -85,B 0,C 180,E1 24978.045,E2 24978.045} C_VEL
LIN {X 0,Y 577.356,Z 501.642,A -85,B 0,C 180,E1 24977.3,E2 24977.3} C_VEL
LIN {X 0,Y 578.731,Z 504.97,A -85,B 0,C 180,E1 24976.809,E2 24976.809} C_VEL
LIN {X 0,Y 586.559,Z 522.264,A -85,B 0,C 180,E1 24974.417,E2 24974.417} C_VEL
LIN {X 0,Y 594.634,Z 541.478,A -85,B 0,C 180,E1 24971.992,E2 24971.992} C_VEL
LIN {X 0,Y 600.861,Z 557.948,A -85,B 0,C 180,E1 24970.089,E2 24970.089} C_VEL
LIN {X 0,Y 597.067,Z 602.75,A -85,B 0,C 180,E1 24966.775,E2 24966.775} C_VEL
LIN {X 0,Y 594.395,Z 639.036,A -85,B 0,C 180,E1 24964.173,E2 24964.173} C_VEL
LIN {X 0,Y 601.931,Z 682.091,A -85,B 0,C 180,E1 24963.031,E2 24963.031} C_VEL
LIN {X 0,Y 601.669,Z 700.04,A -85,B 0,C 180,E1 24962.809,E2 24962.809} C_VEL
LIN {X 0,Y 600.758,Z 707.741,A -85,B 0,C 180,E1 24962.77,E2 24962.77} C_VEL
LIN {X 0,Y 595.412,Z 728.278,A -85,B 0,C 180,E1 24962.873,E2 24962.873} C_VEL
LIN {X 0,Y 594.683,Z 734.889,A -85,B 0,C 180,E1 24962.836,E2 24962.836} C_VEL
LIN {X 0,Y 591.623,Z 954.31,A -85,B 0,C 180,E1 24960.154,E2 24960.154} C_VEL
LIN {X 0,Y 590.637,Z 976.156,A -85,B 0,C 180,E1 24959.732,E2 24959.732} C_VEL
LIN {X 0,Y 589.359,Z 997.123,A -85,B 0,C 180,E1 24959.165,E2 24959.165} C_VEL
LIN {X 0,Y 587.736,Z 1017.199,A -85,B 0,C 180,E1 24958.446,E2 24958.446} C_VEL
LIN {X 0,Y 585.84,Z 1037.307,A -85,B 0,C 180,E1 24957.55,E2 24957.55} C_VEL
LIN {X 0,Y 583.776,Z 1056.719,A -85,B 0,C 180,E1 24956.498,E2 24956.498} C_VEL
LIN {X 0,Y 581.552,Z 1075.176,A -85,B 0,C 180,E1 24955.287,E2 24955.287} C_VEL
LIN {X 0,Y 579.169,Z 1093.996,A -85,B 0,C 180,E1 24953.827,E2 24953.827} C_VEL
LIN {X 0,Y 576.991,Z 1110.69,A -85,B 0,C 180,E1 24952.303,E2 24952.303} C_VEL
LIN {X 0,Y 574.969,Z 1125.791,A -85,B 0,C 180,E1 24950.672,E2 24950.672} C_VEL
LIN {X 0,Y 573.079,Z 1140.426,A -85,B 0,C 180,E1 24948.831,E2 24948.831} C_VEL
LIN {X 0,Y 571.567,Z 1152.988,A -85,B 0,C 180,E1 24946.986,E2 24946.986} C_VEL
LIN {X 0,Y 570.264,Z 1164.674,A -85,B 0,C 180,E1 24944.936,E2 24944.936} C_VEL
LIN {X 0,Y 569.283,Z 1174.93,A -85,B 0,C 180,E1 24942.785,E2 24942.785} C_VEL
LIN {X 0,Y 568.645,Z 1183.363,A -85,B 0,C 180,E1 24940.639,E2 24940.639} C_VEL
LIN {X 0,Y 568.263,Z 1189.991,A -85,B 0,C 180,E1 24938.499,E2 24938.499} C_VEL
LIN {X 0,Y 568.029,Z 1195.485,A -85,B 0,C 180,E1 24936.164,E2 24936.164} C_VEL
LIN {X 0,Y 567.954,Z 1199.125,A -85,B 0,C 180,E1 24933.937,E2 24933.937} C_VEL
LIN {X 0,Y 567.926,Z 1201.094,A -85,B 0,C 180,E1 24931.715,E2 24931.715} C_VEL
LIN {X 0,Y 567.917,Z 1201.519,A -85,B 0,C 180,E1 24929.395,E2 24929.395} C_VEL
LIN {X 0,Y 567.935,Z 1200.416,A -85,B 0,C 180,E1 24927.175,E2 24927.175} C_VEL
LIN {X 0,Y 567.969,Z 1197.782,A -85,B 0,C 180,E1 24925.052,E2 24925.052} C_VEL
LIN {X 0,Y 568.107,Z 1193.296,A -85,B 0,C 180,E1 24922.72,E2 24922.72} C_VEL
LIN {X 0,Y 568.401,Z 1187.356,A -85,B 0,C 180,E1 24920.482,E2 24920.482} C_VEL
LIN {X 0,Y 568.884,Z 1179.892,A -85,B 0,C 180,E1 24918.339,E2 24918.339} C_VEL
LIN {X 0,Y 569.714,Z 1170.224,A -85,B 0,C 180,E1 24916.088,E2 24916.088} C_VEL
LIN {X 0,Y 570.811,Z 1159.609,A -85,B 0,C 180,E1 24914.038,E2 24914.038} C_VEL
LIN {X 0,Y 572.203,Z 1147.528,A -85,B 0,C 180,E1 24912.089,E2 24912.089} C_VEL
LIN {X 0,Y 573.96,Z 1133.54,A -85,B 0,C 180,E1 24910.175,E2 24910.175} C_VEL
LIN {X 0,Y 575.964,Z 1118.379,A -85,B 0,C 180,E1 24908.406,E2 24908.406} C_VEL
LIN {X 0,Y 577.992,Z 1103.029,A -85,B 0,C 180,E1 24906.879,E2 24906.879} C_VEL
LIN {X 0,Y 580.242,Z 1085.727,A -85,B 0,C 180,E1 24905.409,E2 24905.409} C_VEL
LIN {X 0,Y 582.421,Z 1068.415,A -85,B 0,C 180,E1 24904.148,E2 24904.148} C_VEL
LIN {X 0,Y 584.57,Z 1049.381,A -85,B 0,C 180,E1 24902.992,E2 24902.992} C_VEL
LIN {X 0,Y 586.723,Z 1028.498,A -85,B 0,C 180,E1 24901.944,E2 24901.944} C_VEL
LIN {X 0,Y 588.516,Z 1008.449,A -85,B 0,C 180,E1 24901.123,E2 24901.123} C_VEL
LIN {X 0,Y 589.995,Z 987.261,A -85,B 0,C 180,E1 24900.455,E2 24900.455} C_VEL
LIN {X 0,Y 591.224,Z 964.664,A -85,B 0,C 180,E1 24899.933,E2 24899.933} C_VEL
LIN {X 0,Y 591.939,Z 942.471,A -85,B 0,C 180,E1 24899.59,E2 24899.59} C_VEL
LIN {X 0,Y 595.491,Z 682.576,A -85,B 0,C 180,E1 24896.418,E2 24896.418} C_VEL
LIN {X 0,Y 587.556,Z 637.377,A -85,B 0,C 180,E1 24895.17,E2 24895.17} C_VEL
LIN {X 0,Y 591.306,Z 592.028,A -85,B 0,C 180,E1 24891.842,E2 24891.842} C_VEL
LIN {X 0,Y 594.097,Z 561.209,A -85,B 0,C 180,E1 24889.529,E2 24889.529} C_VEL
LIN {X 0,Y 585.71,Z 539.557,A -85,B 0,C 180,E1 24886.942,E2 24886.942} C_VEL
LIN {X 0,Y 577.726,Z 521.13,A -85,B 0,C 180,E1 24884.503,E2 24884.503} C_VEL
LIN {X 0,Y 572.669,Z 509.986,A -85,B 0,C 180,E1 24882.918,E2 24882.918} C_VEL
LIN {X 0,Y 569.429,Z 502.614,A -85,B 0,C 180,E1 24881.81,E2 24881.81} C_VEL
LIN {X 0,Y 569.35,Z 502.299,A -85,B 0,C 180,E1 24880.792,E2 24880.792} C_VEL
LIN {X 0,Y 569.367,Z 502.25,A -85,B 0,C 180,E1 24877.463,E2 24877.463} C_VEL
LIN {X 0,Y 569.374,Z 502.299,A -85,B 0,C 180,E1 24874.192,E2 24874.192} C_VEL
LIN {X 0,Y 569.349,Z 502.301,A -85,B 0,C 180,E1 24870.823,E2 24870.823} C_VEL
LIN {X 0,Y 569.381,Z 502.296,A -85,B 0,C 180,E1 24867.621,E2 24867.621} C_VEL
LIN {X 0,Y 569.348,Z 502.311,A -85,B 0,C 180,E1 24864.375,E2 24864.375} C_VEL
LIN {X 0,Y 569.373,Z 502.305,A -85,B 0,C 180,E1 24860.993,E2 24860.993} C_VEL
LIN {X 0,Y 569.374,Z 502.299,A -85,B 0,C 180,E1 24857.687,E2 24857.687} C_VEL
LIN {X 0,Y 569.344,Z 502.289,A -85,B 0,C 180,E1 24854.441,E2 24854.441} C_VEL
LIN {X 0,Y 569.379,Z 502.29,A -85,B 0,C 180,E1 24851.241,E2 24851.241} C_VEL
LIN {X 0,Y 569.342,Z 502.309,A -85,B 0,C 180,E1 24847.975,E2 24847.975} C_VEL
LIN {X 0,Y 569.377,Z 502.297,A -85,B 0,C 180,E1 24844.734,E2 24844.734} C_VEL
LIN {X 0,Y 569.346,Z 502.292,A -85,B 0,C 180,E1 24841.51,E2 24841.51} C_VEL
LIN {X 0,Y 569.347,Z 502.305,A -85,B 0,C 180,E1 24838.088,E2 24838.088} C_VEL
LIN {X 0,Y 569.379,Z 502.303,A -85,B 0,C 180,E1 24834.862,E2 24834.862} C_VEL
LIN {X 0,Y 569.332,Z 502.287,A -85,B 0,C 180,E1 24831.618,E2 24831.618} C_VEL
LIN {X 0,Y 569.381,Z 502.293,A -85,B 0,C 180,E1 24828.452,E2 24828.452} C_VEL
LIN {X 0,Y 569.334,Z 502.31,A -85,B 0,C 180,E1 24825.247,E2 24825.247} C_VEL
LIN {X 0,Y 569.373,Z 502.3,A -85,B 0,C 180,E1 24821.996,E2 24821.996} C_VEL
LIN {X 0,Y 569.346,Z 502.292,A -85,B 0,C 180,E1 24818.79,E2 24818.79} C_VEL
LIN {X 0,Y 569.34,Z 502.292,A -85,B 0,C 180,E1 24815.403,E2 24815.403} C_VEL
LIN {X 0,Y 569.377,Z 502.295,A -85,B 0,C 180,E1 24812.258,E2 24812.258} C_VEL
LIN {X 0,Y 569.332,Z 502.3,A -85,B 0,C 180,E1 24808.984,E2 24808.984} C_VEL
LIN {X 0,Y 569.375,Z 502.251,A -85,B 0,C 180,E1 24805.802,E2 24805.802} C_VEL
LIN {X 0,Y 569.327,Z 502.286,A -85,B 0,C 180,E1 24802.705,E2 24802.705} C_VEL
LIN {X 0,Y 569.382,Z 502.271,A -85,B 0,C 180,E1 24799.477,E2 24799.477} C_VEL
LIN {X 0,Y 569.379,Z 502.648,A -85,B 0,C 180,E1 24798.543,E2 24798.543} C_VEL
LIN {X 0,Y 570.931,Z 506.164,A -85,B 0,C 180,E1 24798.009,E2 24798.009} C_VEL
LIN {X 0,Y 578.757,Z 522.922,A -85,B 0,C 180,E1 24795.661,E2 24795.661} C_VEL
LIN {X 0,Y 586.955,Z 541.761,A -85,B 0,C 180,E1 24793.259,E2 24793.259} C_VEL
LIN {X 0,Y 600.654,Z 564.266,A -85,B 0,C 180,E1 24791.792,E2 24791.792} C_VEL
LIN {X 0,Y 601.668,Z 566.453,A -85,B 0,C 180,E1 24791.681,E2 24791.681} C_VEL
LIN {X 0,Y 595.647,Z 813.165,A -85,B 0,C 180,E1 24788.239,E2 24788.239} C_VEL
LIN {X 0,Y 593.076,Z 921.439,A -85,B 0,C 180,E1 24786.713,E2 24786.713} C_VEL
LIN {X 0,Y 591.913,Z 946.347,A -85,B 0,C 180,E1 24786.197,E2 24786.197} C_VEL
LIN {X 0,Y 590.658,Z 967.172,A -85,B 0,C 180,E1 24785.63,E2 24785.63} C_VEL
LIN {X 0,Y 588.917,Z 991.784,A -85,B 0,C 180,E1 24784.782,E2 24784.782} C_VEL
LIN {X 0,Y 587.282,Z 1011.658,A -85,B 0,C 180,E1 24783.947,E2 24783.947} C_VEL
LIN {X 0,Y 585.288,Z 1033.992,A -85,B 0,C 180,E1 24782.846,E2 24782.846} C_VEL
LIN {X 0,Y 583.266,Z 1054.654,A -85,B 0,C 180,E1 24781.638,E2 24781.638} C_VEL
LIN {X 0,Y 581.139,Z 1075.911,A -85,B 0,C 180,E1 24780.215,E2 24780.215} C_VEL
LIN {X 0,Y 578.983,Z 1096.235,A -85,B 0,C 180,E1 24778.634,E2 24778.634} C_VEL
LIN {X 0,Y 576.958,Z 1115.929,A -85,B 0,C 180,E1 24776.892,E2 24776.892} C_VEL
LIN {X 0,Y 575.308,Z 1131.492,A -85,B 0,C 180,E1 24775.311,E2 24775.311} C_VEL
LIN {X 0,Y 573.706,Z 1147.18,A -85,B 0,C 180,E1 24773.522,E2 24773.522} C_VEL
LIN {X 0,Y 572.209,Z 1162.263,A -85,B 0,C 180,E1 24771.527,E2 24771.527} C_VEL
LIN {X 0,Y 571.085,Z 1174.077,A -85,B 0,C 180,E1 24769.749,E2 24769.749} C_VEL
LIN {X 0,Y 569.927,Z 1187.672,A -85,B 0,C 180,E1 24767.368,E2 24767.368} C_VEL
LIN {X 0,Y 569.247,Z 1196.863,A -85,B 0,C 180,E1 24765.485,E2 24765.485} C_VEL
LIN {X 0,Y 568.685,Z 1206.012,A -85,B 0,C 180,E1 24763.316,E2 24763.316} C_VEL
LIN {X 0,Y 568.273,Z 1214.104,A -85,B 0,C 180,E1 24760.942,E2 24760.942} C_VEL
LIN {X 0,Y 568.063,Z 1219.992,A -85,B 0,C 180,E1 24758.808,E2 24758.808} C_VEL
LIN {X 0,Y 567.957,Z 1225.174,A -85,B 0,C 180,E1 24756.266,E2 24756.266} C_VEL
LIN {X 0,Y 567.921,Z 1228.121,A -85,B 0,C 180,E1 24754.139,E2 24754.139} C_VEL
LIN {X 0,Y 567.902,Z 1230.038,A -85,B 0,C 180,E1 24751.816,E2 24751.816} C_VEL
LIN {X 0,Y 567.885,Z 1230.37,A -85,B 0,C 180,E1 24749.395,E2 24749.395} C_VEL
LIN {X 0,Y 567.892,Z 1229.493,A -85,B 0,C 180,E1 24747.376,E2 24747.376} C_VEL
LIN {X 0,Y 567.908,Z 1227.211,A -85,B 0,C 180,E1 24745.051,E2 24745.051} C_VEL
LIN {X 0,Y 567.973,Z 1223.308,A -85,B 0,C 180,E1 24742.718,E2 24742.718} C_VEL
LIN {X 0,Y 568.094,Z 1218.955,A -85,B 0,C 180,E1 24740.784,E2 24740.784} C_VEL
LIN {X 0,Y 568.337,Z 1212.436,A -85,B 0,C 180,E1 24738.507,E2 24738.507} C_VEL
LIN {X 0,Y 568.784,Z 1203.936,A -85,B 0,C 180,E1 24736.168,E2 24736.168} C_VEL
LIN {X 0,Y 569.383,Z 1194.99,A -85,B 0,C 180,E1 24734.101,E2 24734.101} C_VEL
LIN {X 0,Y 570.34,Z 1182.707,A -85,B 0,C 180,E1 24731.711,E2 24731.711} C_VEL
LIN {X 0,Y 571.403,Z 1170.781,A -85,B 0,C 180,E1 24729.729,E2 24729.729} C_VEL
LIN {X 0,Y 572.872,Z 1155.379,A -85,B 0,C 180,E1 24727.528,E2 24727.528} C_VEL
LIN {X 0,Y 574.342,Z 1140.955,A -85,B 0,C 180,E1 24725.742,E2 24725.742} C_VEL
LIN {X 0,Y 576.256,Z 1122.403,A -85,B 0,C 180,E1 24723.74,E2 24723.74} C_VEL
LIN {X 0,Y 578.034,Z 1105.536,A -85,B 0,C 180,E1 24722.158,E2 24722.158} C_VEL
LIN {X 0,Y 580.297,Z 1083.599,A -85,B 0,C 180,E1 24720.363,E2 24720.363} C_VEL
LIN {X 0,Y 582.343,Z 1063.955,A -85,B 0,C 180,E1 24718.958,E2 24718.958} C_VEL
LIN {X 0,Y 584.492,Z 1042.379,A -85,B 0,C 180,E1 24717.627,E2 24717.627} C_VEL
LIN {X 0,Y 586.324,Z 1022.717,A -85,B 0,C 180,E1 24716.577,E2 24716.577} C_VEL
LIN {X 0,Y 588.368,Z 998.46,A -85,B 0,C 180,E1 24715.483,E2 24715.483} C_VEL
LIN {X 0,Y 590.001,Z 976.535,A -85,B 0,C 180,E1 24714.669,E2 24714.669} C_VEL
LIN {X 0,Y 591.625,Z 951.336,A -85,B 0,C 180,E1 24713.927,E2 24713.927} C_VEL
LIN {X 0,Y 592.709,Z 930.409,A -85,B 0,C 180,E1 24713.457,E2 24713.457} C_VEL
LIN {X 0,Y 593.659,Z 901.802,A -85,B 0,C 180,E1 24712.993,E2 24712.993} C_VEL
LIN {X 0,Y 599.456,Z 654.843,A -85,B 0,C 180,E1 24709.547,E2 24709.547} C_VEL
LIN {X 0,Y 601.502,Z 565.681,A -85,B 0,C 180,E1 24708.296,E2 24708.296} C_VEL
LIN {X 0,Y 587.16,Z 542.221,A -85,B 0,C 180,E1 24706.791,E2 24706.791} C_VEL
LIN {X 0,Y 579.576,Z 524.868,A -85,B 0,C 180,E1 24704.601,E2 24704.601} C_VEL
LIN {X 0,Y 572.975,Z 510.381,A -85,B 0,C 180,E1 24702.617,E2 24702.617} C_VEL
LIN {X 0,Y 570.494,Z 505.532,A -85,B 0,C 180,E1 24701.895,E2 24701.895} C_VEL
LIN {X 0,Y 569.351,Z 502.461,A -85,B 0,C 180,E1 24701.421,E2 24701.421} C_VEL
LIN {X 0,Y 569.381,Z 502.252,A -85,B 0,C 180,E1 24698.309,E2 24698.309} C_VEL
LIN {X 0,Y 569.328,Z 502.284,A -85,B 0,C 180,E1 24695.174,E2 24695.174} C_VEL
LIN {X 0,Y 569.376,Z 502.265,A -85,B 0,C 180,E1 24691.91,E2 24691.91} C_VEL
LIN {X 0,Y 569.338,Z 502.296,A -85,B 0,C 180,E1 24688.764,E2 24688.764} C_VEL
LIN {X 0,Y 569.351,Z 502.294,A -85,B 0,C 180,E1 24685.373,E2 24685.373} C_VEL
LIN {X 0,Y 569.373,Z 502.305,A -85,B 0,C 180,E1 24682.183,E2 24682.183} C_VEL
LIN {X 0,Y 569.338,Z 502.31,A -85,B 0,C 180,E1 24678.853,E2 24678.853} C_VEL
LIN {X 0,Y 569.383,Z 502.298,A -85,B 0,C 180,E1 24675.586,E2 24675.586} C_VEL
LIN {X 0,Y 569.338,Z 502.29,A -85,B 0,C 180,E1 24672.372,E2 24672.372} C_VEL
LIN {X 0,Y 569.372,Z 502.292,A -85,B 0,C 180,E1 24669.094,E2 24669.094} C_VEL
LIN {X 0,Y 569.361,Z 502.304,A -85,B 0,C 180,E1 24665.846,E2 24665.846} C_VEL
LIN {X 0,Y 569.346,Z 502.298,A -85,B 0,C 180,E1 24662.516,E2 24662.516} C_VEL
LIN {X 0,Y 569.381,Z 502.288,A -85,B 0,C 180,E1 24659.296,E2 24659.296} C_VEL
LIN {X 0,Y 569.342,Z 502.307,A -85,B 0,C 180,E1 24656.073,E2 24656.073} C_VEL
LIN {X 0,Y 569.382,Z 502.296,A -85,B 0,C 180,E1 24652.821,E2 24652.821} C_VEL
LIN {X 0,Y 569.351,Z 502.286,A -85,B 0,C 180,E1 24649.557,E2 24649.557} C_VEL
LIN {X 0,Y 569.362,Z 502.295,A -85,B 0,C 180,E1 24646.182,E2 24646.182} C_VEL
LIN {X 0,Y 569.38,Z 502.305,A -85,B 0,C 180,E1 24642.946,E2 24642.946} C_VEL
LIN {X 0,Y 569.349,Z 502.308,A -85,B 0,C 180,E1 24639.652,E2 24639.652} C_VEL
LIN {X 0,Y 569.377,Z 502.29,A -85,B 0,C 180,E1 24636.397,E2 24636.397} C_VEL
LIN {X 0,Y 569.355,Z 502.292,A -85,B 0,C 180,E1 24633.139,E2 24633.139} C_VEL
LIN {X 0,Y 569.374,Z 502.294,A -85,B 0,C 180,E1 24629.767,E2 24629.767} C_VEL
LIN {X 0,Y 569.377,Z 502.292,A -85,B 0,C 180,E1 24626.415,E2 24626.415} C_VEL
LIN {X 0,Y 569.349,Z 502.264,A -85,B 0,C 180,E1 24623.207,E2 24623.207} C_VEL
LIN {X 0,Y 569.374,Z 502.296,A -85,B 0,C 180,E1 24619.964,E2 24619.964} C_VEL
LIN {X 0,Y 569.405,Z 502.481,A -85,B 0,C 180,E1 24618.119,E2 24618.119} C_VEL
LIN {X 0,Y 570.755,Z 505.868,A -85,B 0,C 180,E1 24617.587,E2 24617.587} C_VEL
LIN {X 0,Y 577.469,Z 520.574,A -85,B 0,C 180,E1 24615.472,E2 24615.472} C_VEL
LIN {X 0,Y 584.537,Z 536.827,A -85,B 0,C 180,E1 24613.308,E2 24613.308} C_VEL
LIN {X 0,Y 592.295,Z 556.501,A -85,B 0,C 180,E1 24610.918,E2 24610.918} C_VEL
LIN {X 0,Y 594.049,Z 561.543,A -85,B 0,C 180,E1 24610.349,E2 24610.349} C_VEL
LIN {X 0,Y 590.115,Z 605.642,A -85,B 0,C 180,E1 24607.054,E2 24607.054} C_VEL
LIN {X 0,Y 587.587,Z 638.141,A -85,B 0,C 180,E1 24604.701,E2 24604.701} C_VEL
LIN {X 0,Y 595.49,Z 683.353,A -85,B 0,C 180,E1 24603.475,E2 24603.475} C_VEL
LIN {X 0,Y 594.683,Z 734.889,A -85,B 0,C 180,E1 24602.836,E2 24602.836} C_VEL
LIN {X 0,Y 593.726,Z 742.594,A -85,B 0,C 180,E1 24602.8,E2 24602.8} C_VEL
LIN {X 0,Y 588.36,Z 763.127,A -85,B 0,C 180,E1 24602.91,E2 24602.91} C_VEL
LIN {X 0,Y 587.698,Z 769.733,A -85,B 0,C 180,E1 24602.869,E2 24602.869} C_VEL
LIN {X 0,Y 584.985,Z 954.145,A -85,B 0,C 180,E1 24600.593,E2 24600.593} C_VEL
LIN {X 0,Y 583.947,Z 976.005,A -85,B 0,C 180,E1 24600.168,E2 24600.168} C_VEL
LIN {X 0,Y 582.583,Z 997.278,A -85,B 0,C 180,E1 24599.586,E2 24599.586} C_VEL
LIN {X 0,Y 580.909,Z 1017.166,A -85,B 0,C 180,E1 24598.868,E2 24598.868} C_VEL
LIN {X 0,Y 578.808,Z 1038.271,A -85,B 0,C 180,E1 24597.913,E2 24597.913} C_VEL
LIN {X 0,Y 576.656,Z 1057.554,A -85,B 0,C 180,E1 24596.851,E2 24596.851} C_VEL
LIN {X 0,Y 574.342,Z 1075.827,A -85,B 0,C 180,E1 24595.633,E2 24595.633} C_VEL
LIN {X 0,Y 571.833,Z 1094.615,A -85,B 0,C 180,E1 24594.152,E2 24594.152} C_VEL
LIN {X 0,Y 569.55,Z 1111.232,A -85,B 0,C 180,E1 24592.61,E2 24592.61} C_VEL
LIN {X 0,Y 567.395,Z 1126.525,A -85,B 0,C 180,E1 24590.933,E2 24590.933} C_VEL
LIN {X 0,Y 565.431,Z 1140.884,A -85,B 0,C 180,E1 24589.095,E2 24589.095} C_VEL
LIN {X 0,Y 563.832,Z 1153.415,A -85,B 0,C 180,E1 24587.226,E2 24587.226} C_VEL
LIN {X 0,Y 562.442,Z 1165.162,A -85,B 0,C 180,E1 24585.131,E2 24585.131} C_VEL
LIN {X 0,Y 561.405,Z 1175.289,A -85,B 0,C 180,E1 24582.968,E2 24582.968} C_VEL
LIN {X 0,Y 560.714,Z 1183.688,A -85,B 0,C 180,E1 24580.791,E2 24580.791} C_VEL
LIN {X 0,Y 560.286,Z 1190.585,A -85,B 0,C 180,E1 24578.518,E2 24578.518} C_VEL
LIN {X 0,Y 560.047,Z 1195.751,A -85,B 0,C 180,E1 24576.252,E2 24576.252} C_VEL
LIN {X 0,Y 559.962,Z 1199.354,A -85,B 0,C 180,E1 24573.993,E2 24573.993} C_VEL
LIN {X 0,Y 559.934,Z 1201.24,A -85,B 0,C 180,E1 24571.842,E2 24571.842} C_VEL
LIN {X 0,Y 559.919,Z 1201.746,A -85,B 0,C 180,E1 24569.488,E2 24569.488} C_VEL
LIN {X 0,Y 559.938,Z 1200.717,A -85,B 0,C 180,E1 24567.237,E2 24567.237} C_VEL
LIN {X 0,Y 559.979,Z 1198.028,A -85,B 0,C 180,E1 24564.981,E2 24564.981} C_VEL
LIN {X 0,Y 560.134,Z 1193.58,A -85,B 0,C 180,E1 24562.616,E2 24562.616} C_VEL
LIN {X 0,Y 560.451,Z 1187.666,A -85,B 0,C 180,E1 24560.346,E2 24560.346} C_VEL
LIN {X 0,Y 560.973,Z 1180.229,A -85,B 0,C 180,E1 24558.172,E2 24558.172} C_VEL
LIN {X 0,Y 561.864,Z 1170.597,A -85,B 0,C 180,E1 24555.889,E2 24555.889} C_VEL
LIN {X 0,Y 563.034,Z 1160.02,A -85,B 0,C 180,E1 24553.811,E2 24553.811} C_VEL
LIN {X 0,Y 564.505,Z 1147.955,A -85,B 0,C 180,E1 24551.836,E2 24551.836} C_VEL
LIN {X 0,Y 566.324,Z 1134.29,A -85,B 0,C 180,E1 24549.933,E2 24549.933} C_VEL
LIN {X 0,Y 568.414,Z 1119.406,A -85,B 0,C 180,E1 24548.159,E2 24548.159} C_VEL
LIN {X 0,Y 570.601,Z 1103.595,A -85,B 0,C 180,E1 24546.561,E2 24546.561} C_VEL
LIN {X 0,Y 572.966,Z 1086.381,A -85,B 0,C 180,E1 24545.075,E2 24545.075} C_VEL
LIN {X 0,Y 575.239,Z 1069.149,A -85,B 0,C 180,E1 24543.801,E2 24543.801} C_VEL
LIN {X 0,Y 577.487,Z 1050.232,A -85,B 0,C 180,E1 24542.633,E2 24542.633} C_VEL
LIN {X 0,Y 579.739,Z 1029.568,A -85,B 0,C 180,E1 24541.575,E2 24541.575} C_VEL
LIN {X 0,Y 581.545,Z 1010.342,A -85,B 0,C 180,E1 24540.772,E2 24540.772} C_VEL
LIN {X 0,Y 583.133,Z 989.166,A -85,B 0,C 180,E1 24540.08,E2 24540.08} C_VEL
LIN {X 0,Y 584.444,Z 967.372,A -85,B 0,C 180,E1 24539.549,E2 24539.549} C_VEL
LIN {X 0,Y 585.233,Z 945.939,A -85,B 0,C 180,E1 24539.199,E2 24539.199} C_VEL
LIN {X 0,Y 589.082,Z 683.971,A -85,B 0,C 180,E1 24535.965,E2 24535.965} C_VEL
LIN {X 0,Y 580.799,Z 636.488,A -85,B 0,C 180,E1 24534.63,E2 24534.63} C_VEL
LIN {X 0,Y 584.94,Z 589.611,A -85,B 0,C 180,E1 24531.147,E2 24531.147} C_VEL
LIN {X 0,Y 587.297,Z 564.726,A -85,B 0,C 180,E1 24529.256,E2 24529.256} C_VEL
LIN {X 0,Y 579.346,Z 544.014,A -85,B 0,C 180,E1 24526.747,E2 24526.747} C_VEL
LIN {X 0,Y 571.554,Z 525.878,A -85,B 0,C 180,E1 24524.317,E2 24524.317} C_VEL
LIN {X 0,Y 565.162,Z 511.561,A -85,B 0,C 180,E1 24522.245,E2 24522.245} C_VEL
LIN {X 0,Y 561.466,Z 503.669,A -85,B 0,C 180,E1 24521.002,E2 24521.002} C_VEL
LIN {X 0,Y 561.442,Z 503.289,A -85,B 0,C 180,E1 24520.143,E2 24520.143} C_VEL
LIN {X 0,Y 561.404,Z 503.247,A -85,B 0,C 180,E1 24516.886,E2 24516.886} C_VEL
LIN {X 0,Y 561.442,Z 503.281,A -85,B 0,C 180,E1 24513.633,E2 24513.633} C_VEL
LIN {X 0,Y 561.416,Z 503.285,A -85,B 0,C 180,E1 24510.385,E2 24510.385} C_VEL
LIN {X 0,Y 561.421,Z 503.28,A -85,B 0,C 180,E1 24507.011,E2 24507.011} C_VEL
LIN {X 0,Y 561.442,Z 503.28,A -85,B 0,C 180,E1 24503.734,E2 24503.734} C_VEL
LIN {X 0,Y 561.406,Z 503.298,A -85,B 0,C 180,E1 24500.432,E2 24500.432} C_VEL
LIN {X 0,Y 561.442,Z 503.294,A -85,B 0,C 180,E1 24497.089,E2 24497.089} C_VEL
LIN {X 0,Y 561.415,Z 503.283,A -85,B 0,C 180,E1 24493.807,E2 24493.807} C_VEL
LIN {X 0,Y 561.411,Z 503.274,A -85,B 0,C 180,E1 24490.467,E2 24490.467} C_VEL
LIN {X 0,Y 561.446,Z 503.287,A -85,B 0,C 180,E1 24487.264,E2 24487.264} C_VEL
LIN {X 0,Y 561.401,Z 503.295,A -85,B 0,C 180,E1 24483.983,E2 24483.983} C_VEL
LIN {X 0,Y 561.443,Z 503.276,A -85,B 0,C 180,E1 24480.714,E2 24480.714} C_VEL
LIN {X 0,Y 561.404,Z 503.287,A -85,B 0,C 180,E1 24477.448,E2 24477.448} C_VEL
LIN {X 0,Y 561.414,Z 503.296,A -85,B 0,C 180,E1 24474.071,E2 24474.071} C_VEL
LIN {X 0,Y 561.432,Z 503.281,A -85,B 0,C 180,E1 24470.88,E2 24470.88} C_VEL
LIN {X 0,Y 561.396,Z 503.279,A -85,B 0,C 180,E1 24467.554,E2 24467.554} C_VEL
LIN {X 0,Y 561.445,Z 503.284,A -85,B 0,C 180,E1 24464.294,E2 24464.294} C_VEL
LIN {X 0,Y 561.4,Z 503.299,A -85,B 0,C 180,E1 24461.034,E2 24461.034} C_VEL
LIN {X 0,Y 561.422,Z 503.295,A -85,B 0,C 180,E1 24457.706,E2 24457.706} C_VEL
LIN {X 0,Y 561.422,Z 503.283,A -85,B 0,C 180,E1 24454.469,E2 24454.469} C_VEL
LIN {X 0,Y 561.393,Z 503.286,A -85,B 0,C 180,E1 24451.14,E2 24451.14} C_VEL
LIN {X 0,Y 561.44,Z 503.247,A -85,B 0,C 180,E1 24447.962,E2 24447.962} C_VEL
LIN {X 0,Y 561.388,Z 503.274,A -85,B 0,C 180,E1 24444.755,E2 24444.755} C_VEL
LIN {X 0,Y 561.442,Z 503.238,A -85,B 0,C 180,E1 24441.571,E2 24441.571} C_VEL
LIN {X 0,Y 561.469,Z 503.496,A -85,B 0,C 180,E1 24439.391,E2 24439.391} C_VEL
LIN {X 0,Y 562.664,Z 506.716,A -85,B 0,C 180,E1 24438.889,E2 24438.889} C_VEL
LIN {X 0,Y 567.475,Z 516.504,A -85,B 0,C 180,E1 24437.421,E2 24437.421} C_VEL
LIN {X 0,Y 574.718,Z 532.46,A -85,B 0,C 180,E1 24435.22,E2 24435.22} C_VEL
LIN {X 0,Y 579.589,Z 543.612,A -85,B 0,C 180,E1 24433.817,E2 24433.817} C_VEL
LIN {X 0,Y 593.893,Z 566.637,A -85,B 0,C 180,E1 24432.272,E2 24432.272} C_VEL
LIN {X 0,Y 595.314,Z 569.523,A -85,B 0,C 180,E1 24432.116,E2 24432.116} C_VEL
LIN {X 0,Y 589.039,Z 814.548,A -85,B 0,C 180,E1 24428.663,E2 24428.663} C_VEL
LIN {X 0,Y 586.356,Z 921.66,A -85,B 0,C 180,E1 24427.135,E2 24427.135} C_VEL
LIN {X 0,Y 585.144,Z 946.455,A -85,B 0,C 180,E1 24426.616,E2 24426.616} C_VEL
LIN {X 0,Y 583.825,Z 967.393,A -85,B 0,C 180,E1 24426.04,E2 24426.04} C_VEL
LIN {X 0,Y 581.987,Z 992.074,A -85,B 0,C 180,E1 24425.178,E2 24425.178} C_VEL
LIN {X 0,Y 580.205,Z 1012.684,A -85,B 0,C 180,E1 24424.299,E2 24424.299} C_VEL
LIN {X 0,Y 578.011,Z 1035.687,A -85,B 0,C 180,E1 24423.136,E2 24423.136} C_VEL
LIN {X 0,Y 575.907,Z 1056.115,A -85,B 0,C 180,E1 24421.915,E2 24421.915} C_VEL
LIN {X 0,Y 573.5,Z 1078.394,A -85,B 0,C 180,E1 24420.371,E2 24420.371} C_VEL
LIN {X 0,Y 571.403,Z 1097.041,A -85,B 0,C 180,E1 24418.878,E2 24418.878} C_VEL
LIN {X 0,Y 569.182,Z 1117.094,A -85,B 0,C 180,E1 24417.044,E2 24417.044} C_VEL
LIN {X 0,Y 567.391,Z 1133.367,A -85,B 0,C 180,E1 24415.354,E2 24415.354} C_VEL
LIN {X 0,Y 565.575,Z 1150.412,A -85,B 0,C 180,E1 24413.328,E2 24413.328} C_VEL
LIN {X 0,Y 564.297,Z 1162.923,A -85,B 0,C 180,E1 24411.626,E2 24411.626} C_VEL
LIN {X 0,Y 563.037,Z 1176.055,A -85,B 0,C 180,E1 24409.611,E2 24409.611} C_VEL
LIN {X 0,Y 561.949,Z 1188.338,A -85,B 0,C 180,E1 24407.393,E2 24407.393} C_VEL
LIN {X 0,Y 561.19,Z 1198.332,A -85,B 0,C 180,E1 24405.289,E2 24405.289} C_VEL
LIN {X 0,Y 560.589,Z 1207.881,A -85,B 0,C 180,E1 24402.882,E2 24402.882} C_VEL
LIN {X 0,Y 560.259,Z 1214.674,A -85,B 0,C 180,E1 24400.8,E2 24400.8} C_VEL
LIN {X 0,Y 560.058,Z 1220.993,A -85,B 0,C 180,E1 24398.418,E2 24398.418} C_VEL
LIN {X 0,Y 559.951,Z 1225.508,A -85,B 0,C 180,E1 24396.047,E2 24396.047} C_VEL
LIN {X 0,Y 559.916,Z 1228.376,A -85,B 0,C 180,E1 24393.891,E2 24393.891} C_VEL
LIN {X 0,Y 559.903,Z 1230.162,A -85,B 0,C 180,E1 24391.33,E2 24391.33} C_VEL
LIN {X 0,Y 559.889,Z 1230.278,A -85,B 0,C 180,E1 24389.181,E2 24389.181} C_VEL
LIN {X 0,Y 559.887,Z 1229.222,A -85,B 0,C 180,E1 24387.031,E2 24387.031} C_VEL
LIN {X 0,Y 559.911,Z 1226.486,A -85,B 0,C 180,E1 24384.569,E2 24384.569} C_VEL
LIN {X 0,Y 559.974,Z 1222.688,A -85,B 0,C 180,E1 24382.407,E2 24382.407} C_VEL
LIN {X 0,Y 560.139,Z 1217.892,A -85,B 0,C 180,E1 24380.341,E2 24380.341} C_VEL
LIN {X 0,Y 560.458,Z 1210.436,A -85,B 0,C 180,E1 24377.848,E2 24377.848} C_VEL
LIN {X 0,Y 560.892,Z 1202.708,A -85,B 0,C 180,E1 24375.759,E2 24375.759} C_VEL
LIN {X 0,Y 561.622,Z 1192.613,A -85,B 0,C 180,E1 24373.45,E2 24373.45} C_VEL
LIN {X 0,Y 562.53,Z 1181.503,A -85,B 0,C 180,E1 24371.335,E2 24371.335} C_VEL
LIN {X 0,Y 563.673,Z 1169.409,A -85,B 0,C 180,E1 24369.33,E2 24369.33} C_VEL
LIN {X 0,Y 565.169,Z 1154.352,A -85,B 0,C 180,E1 24367.183,E2 24367.183} C_VEL
LIN {X 0,Y 566.769,Z 1139.24,A -85,B 0,C 180,E1 24365.308,E2 24365.308} C_VEL
LIN {X 0,Y 568.72,Z 1121.212,A -85,B 0,C 180,E1 24363.365,E2 24363.365} C_VEL
LIN {X 0,Y 570.794,Z 1102.636,A -85,B 0,C 180,E1 24361.603,E2 24361.603} C_VEL
LIN {X 0,Y 573.029,Z 1082.424,A -85,B 0,C 180,E1 24359.938,E2 24359.938} C_VEL
LIN {X 0,Y 575.325,Z 1061.929,A -85,B 0,C 180,E1 24358.459,E2 24358.459} C_VEL
LIN {X 0,Y 577.546,Z 1040.319,A -85,B 0,C 180,E1 24357.13,E2 24357.13} C_VEL
LIN {X 0,Y 579.69,Z 1018.421,A -85,B 0,C 180,E1 24355.965,E2 24355.965} C_VEL
LIN {X 0,Y 581.682,Z 995.568,A -85,B 0,C 180,E1 24354.962,E2 24354.962} C_VEL
LIN {X 0,Y 583.48,Z 972.68,A -85,B 0,C 180,E1 24354.123,E2 24354.123} C_VEL
LIN {X 0,Y 584.974,Z 949.262,A -85,B 0,C 180,E1 24353.455,E2 24353.455} C_VEL
LIN {X 0,Y 586.119,Z 927.641,A -85,B 0,C 180,E1 24352.977,E2 24352.977} C_VEL
LIN {X 0,Y 587.172,Z 893.172,A -85,B 0,C 180,E1 24352.444,E2 24352.444} C_VEL
LIN {X 0,Y 593.255,Z 647.706,A -85,B 0,C 180,E1 24348.98,E2 24348.98} C_VEL
LIN {X 0,Y 595.149,Z 568.863,A -85,B 0,C 180,E1 24347.863,E2 24347.863} C_VEL
LIN {X 0,Y 580.603,Z 545.25,A -85,B 0,C 180,E1 24346.311,E2 24346.311} C_VEL
LIN {X 0,Y 578.996,Z 542.389,A -85,B 0,C 180,E1 24346.066,E2 24346.066} C_VEL
LIN {X 0,Y 570.549,Z 523.151,A -85,B 0,C 180,E1 24343.53,E2 24343.53} C_VEL
LIN {X 0,Y 564.666,Z 510.812,A -85,B 0,C 180,E1 24341.745,E2 24341.745} C_VEL
LIN {X 0,Y 561.488,Z 503.641,A -85,B 0,C 180,E1 24340.66,E2 24340.66} C_VEL
LIN {X 0,Y 561.399,Z 503.244,A -85,B 0,C 180,E1 24339.748,E2 24339.748} C_VEL
LIN {X 0,Y 561.437,Z 503.296,A -85,B 0,C 180,E1 24336.501,E2 24336.501} C_VEL
LIN {X 0,Y 561.387,Z 503.235,A -85,B 0,C 180,E1 24333.166,E2 24333.166} C_VEL
LIN {X 0,Y 561.445,Z 503.295,A -85,B 0,C 180,E1 24329.856,E2 24329.856} C_VEL
LIN {X 0,Y 561.405,Z 503.299,A -85,B 0,C 180,E1 24326.668,E2 24326.668} C_VEL
LIN {X 0,Y 561.408,Z 503.302,A -85,B 0,C 180,E1 24323.222,E2 24323.222} C_VEL
LIN {X 0,Y 561.439,Z 503.284,A -85,B 0,C 180,E1 24319.995,E2 24319.995} C_VEL
LIN {X 0,Y 561.397,Z 503.281,A -85,B 0,C 180,E1 24316.664,E2 24316.664} C_VEL
LIN {X 0,Y 561.441,Z 503.28,A -85,B 0,C 180,E1 24313.387,E2 24313.387} C_VEL
LIN {X 0,Y 561.41,Z 503.296,A -85,B 0,C 180,E1 24310.156,E2 24310.156} C_VEL
LIN {X 0,Y 561.413,Z 503.289,A -85,B 0,C 180,E1 24306.751,E2 24306.751} C_VEL
LIN {X 0,Y 561.437,Z 503.272,A -85,B 0,C 180,E1 24303.472,E2 24303.472} C_VEL
LIN {X 0,Y 561.402,Z 503.29,A -85,B 0,C 180,E1 24300.204,E2 24300.204} C_VEL
LIN {X 0,Y 561.442,Z 503.293,A -85,B 0,C 180,E1 24296.937,E2 24296.937} C_VEL
LIN {X 0,Y 561.416,Z 503.28,A -85,B 0,C 180,E1 24293.601,E2 24293.601} C_VEL
LIN {X 0,Y 561.412,Z 503.277,A -85,B 0,C 180,E1 24290.155,E2 24290.155} C_VEL
LIN {X 0,Y 561.442,Z 503.296,A -85,B 0,C 180,E1 24286.823,E2 24286.823} C_VEL
LIN {X 0,Y 561.41,Z 503.297,A -85,B 0,C 180,E1 24283.55,E2 24283.55} C_VEL
LIN {X 0,Y 561.438,Z 503.28,A -85,B 0,C 180,E1 24280.222,E2 24280.222} C_VEL
LIN {X 0,Y 561.434,Z 503.275,A -85,B 0,C 180,E1 24276.933,E2 24276.933} C_VEL
LIN {X 0,Y 561.416,Z 503.281,A -85,B 0,C 180,E1 24273.56,E2 24273.56} C_VEL
LIN {X 0,Y 561.439,Z 503.285,A -85,B 0,C 180,E1 24270.323,E2 24270.323} C_VEL
LIN {X 0,Y 561.415,Z 503.286,A -85,B 0,C 180,E1 24267.017,E2 24267.017} C_VEL
LIN {X 0,Y 561.431,Z 503.259,A -85,B 0,C 180,E1 24263.625,E2 24263.625} C_VEL
LIN {X 0,Y 561.44,Z 503.269,A -85,B 0,C 180,E1 24260.256,E2 24260.256} C_VEL
LIN {X 0,Y 561.453,Z 503.554,A -85,B 0,C 180,E1 24258.917,E2 24258.917} C_VEL
LIN {X 0,Y 562.886,Z 506.964,A -85,B 0,C 180,E1 24258.366,E2 24258.366} C_VEL
LIN {X 0,Y 569.194,Z 520.482,A -85,B 0,C 180,E1 24256.34,E2 24256.34} C_VEL
LIN {X 0,Y 577.013,Z 538.462,A -85,B 0,C 180,E1 24253.873,E2 24253.873} C_VEL
LIN {X 0,Y 585.156,Z 558.939,A -85,B 0,C 180,E1 24251.323,E2 24251.323} C_VEL
LIN {X 0,Y 587.264,Z 564.968,A -85,B 0,C 180,E1 24250.628,E2 24250.628} C_VEL
LIN {X 0,Y 583.209,Z 608.193,A -85,B 0,C 180,E1 24247.366,E2 24247.366} C_VEL
LIN {X 0,Y 580.829,Z 637.291,A -85,B 0,C 180,E1 24245.24,E2 24245.24} C_VEL
LIN {X 0,Y 589.086,Z 684.608,A -85,B 0,C 180,E1 24243.928,E2 24243.928} C_VEL
LIN {X 0,Y 587.698,Z 769.733,A -85,B 0,C 180,E1 24242.869,E2 24242.869} C_VEL
LIN {X 0,Y 586.819,Z 777.434,A -85,B 0,C 180,E1 24242.828,E2 24242.828} C_VEL
LIN {X 0,Y 581.435,Z 797.967,A -85,B 0,C 180,E1 24242.941,E2 24242.941} C_VEL
LIN {X 0,Y 580.725,Z 804.58,A -85,B 0,C 180,E1 24242.904,E2 24242.904} C_VEL
LIN {X 0,Y 578.371,Z 954.13,A -85,B 0,C 180,E1 24241.039,E2 24241.039} C_VEL
LIN {X 0,Y 577.282,Z 975.928,A -85,B 0,C 180,E1 24240.611,E2 24240.611} C_VEL
LIN {X 0,Y 575.868,Z 996.995,A -85,B 0,C 180,E1 24240.032,E2 24240.032} C_VEL
LIN {X 0,Y 574.11,Z 1017.09,A -85,B 0,C 180,E1 24239.3,E2 24239.3} C_VEL
LIN {X 0,Y 571.907,Z 1038.209,A -85,B 0,C 180,E1 24238.337,E2 24238.337} C_VEL
LIN {X 0,Y 569.655,Z 1057.508,A -85,B 0,C 180,E1 24237.265,E2 24237.265} C_VEL
LIN {X 0,Y 567.235,Z 1075.798,A -85,B 0,C 180,E1 24236.034,E2 24236.034} C_VEL
LIN {X 0,Y 564.597,Z 1094.607,A -85,B 0,C 180,E1 24234.537,E2 24234.537} C_VEL
LIN {X 0,Y 562.201,Z 1111.247,A -85,B 0,C 180,E1 24232.978,E2 24232.978} C_VEL
LIN {X 0,Y 559.892,Z 1126.783,A -85,B 0,C 180,E1 24231.255,E2 24231.255} C_VEL
LIN {X 0,Y 557.791,Z 1141.307,A -85,B 0,C 180,E1 24229.367,E2 24229.367} C_VEL
LIN {X 0,Y 556.101,Z 1153.799,A -85,B 0,C 180,E1 24227.473,E2 24227.473} C_VEL
LIN {X 0,Y 554.701,Z 1164.884,A -85,B 0,C 180,E1 24225.472,E2 24225.472} C_VEL
LIN {X 0,Y 553.571,Z 1175.176,A -85,B 0,C 180,E1 24223.261,E2 24223.261} C_VEL
LIN {X 0,Y 552.816,Z 1183.643,A -85,B 0,C 180,E1 24221.053,E2 24221.053} C_VEL
LIN {X 0,Y 552.337,Z 1190.57,A -85,B 0,C 180,E1 24218.746,E2 24218.746} C_VEL
LIN {X 0,Y 552.074,Z 1195.799,A -85,B 0,C 180,E1 24216.447,E2 24216.447} C_VEL
LIN {X 0,Y 551.974,Z 1199.467,A -85,B 0,C 180,E1 24214.155,E2 24214.155} C_VEL
LIN {X 0,Y 551.937,Z 1201.449,A -85,B 0,C 180,E1 24211.869,E2 24211.869} C_VEL
LIN {X 0,Y 551.922,Z 1201.951,A -85,B 0,C 180,E1 24209.481,E2 24209.481} C_VEL
LIN {X 0,Y 551.943,Z 1200.928,A -85,B 0,C 180,E1 24207.196,E2 24207.196} C_VEL
LIN {X 0,Y 551.99,Z 1198.257,A -85,B 0,C 180,E1 24204.908,E2 24204.908} C_VEL
LIN {X 0,Y 552.158,Z 1193.835,A -85,B 0,C 180,E1 24202.509,E2 24202.509} C_VEL
LIN {X 0,Y 552.501,Z 1187.942,A -85,B 0,C 180,E1 24200.206,E2 24200.206} C_VEL
LIN {X 0,Y 553.071,Z 1180.456,A -85,B 0,C 180,E1 24197.98,E2 24197.98} C_VEL
LIN {X 0,Y 554.015,Z 1170.933,A -85,B 0,C 180,E1 24195.685,E2 24195.685} C_VEL
LIN {X 0,Y 555.263,Z 1160.395,A -85,B 0,C 180,E1 24193.578,E2 24193.578} C_VEL
LIN {X 0,Y 556.814,Z 1148.352,A -85,B 0,C 180,E1 24191.577,E2 24191.577} C_VEL
LIN {X 0,Y 558.806,Z 1134.198,A -85,B 0,C 180,E1 24189.579,E2 24189.579} C_VEL
LIN {X 0,Y 561.003,Z 1119.417,A -85,B 0,C 180,E1 24187.8,E2 24187.8} C_VEL
LIN {X 0,Y 563.305,Z 1103.592,A -85,B 0,C 180,E1 24186.184,E2 24186.184} C_VEL
LIN {X 0,Y 565.79,Z 1086.353,A -85,B 0,C 180,E1 24184.681,E2 24184.681} C_VEL
LIN {X 0,Y 568.271,Z 1068.356,A -85,B 0,C 180,E1 24183.342,E2 24183.342} C_VEL
LIN {X 0,Y 570.615,Z 1049.509,A -85,B 0,C 180,E1 24182.177,E2 24182.177} C_VEL
LIN {X 0,Y 572.886,Z 1029.482,A -85,B 0,C 180,E1 24181.146,E2 24181.146} C_VEL
LIN {X 0,Y 574.771,Z 1010.242,A -85,B 0,C 180,E1 24180.336,E2 24180.336} C_VEL
LIN {X 0,Y 576.438,Z 989.056,A -85,B 0,C 180,E1 24179.638,E2 24179.638} C_VEL
LIN {X 0,Y 577.809,Z 967.291,A -85,B 0,C 180,E1 24179.104,E2 24179.104} C_VEL
LIN {X 0,Y 578.632,Z 945.859,A -85,B 0,C 180,E1 24178.75,E2 24178.75} C_VEL
LIN {X 0,Y 582.703,Z 685.311,A -85,B 0,C 180,E1 24175.501,E2 24175.501} C_VEL
LIN {X 0,Y 574.093,Z 635.701,A -85,B 0,C 180,E1 24174.082,E2 24174.082} C_VEL
LIN {X 0,Y 578.314,Z 590.419,A -85,B 0,C 180,E1 24170.68,E2 24170.68} C_VEL
LIN {X 0,Y 580.516,Z 568.228,A -85,B 0,C 180,E1 24168.975,E2 24168.975} C_VEL
LIN {X 0,Y 572.99,Z 548.471,A -85,B 0,C 180,E1 24166.547,E2 24166.547} C_VEL
LIN {X 0,Y 565.162,Z 530.099,A -85,B 0,C 180,E1 24164.051,E2 24164.051} C_VEL
LIN {X 0,Y 558.893,Z 516.205,A -85,B 0,C 180,E1 24161.998,E2 24161.998} C_VEL
LIN {X 0,Y 554.621,Z 507.502,A -85,B 0,C 180,E1 24160.604,E2 24160.604} C_VEL
LIN {X 0,Y 553.525,Z 504.447,A -85,B 0,C 180,E1 24160.084,E2 24160.084} C_VEL
LIN {X 0,Y 553.466,Z 504.234,A -85,B 0,C 180,E1 24156.842,E2 24156.842} C_VEL
LIN {X 0,Y 553.502,Z 504.269,A -85,B 0,C 180,E1 24153.558,E2 24153.558} C_VEL
LIN {X 0,Y 553.483,Z 504.271,A -85,B 0,C 180,E1 24150.267,E2 24150.267} C_VEL
LIN {X 0,Y 553.473,Z 504.269,A -85,B 0,C 180,E1 24146.849,E2 24146.849} C_VEL
LIN {X 0,Y 553.503,Z 504.266,A -85,B 0,C 180,E1 24143.53,E2 24143.53} C_VEL
LIN {X 0,Y 553.468,Z 504.284,A -85,B 0,C 180,E1 24140.296,E2 24140.296} C_VEL
LIN {X 0,Y 553.494,Z 504.283,A -85,B 0,C 180,E1 24136.909,E2 24136.909} C_VEL
LIN {X 0,Y 553.495,Z 504.273,A -85,B 0,C 180,E1 24133.583,E2 24133.583} C_VEL
LIN {X 0,Y 553.464,Z 504.264,A -85,B 0,C 180,E1 24130.198,E2 24130.198} C_VEL
LIN {X 0,Y 553.504,Z 504.271,A -85,B 0,C 180,E1 24126.952,E2 24126.952} C_VEL
LIN {X 0,Y 553.469,Z 504.287,A -85,B 0,C 180,E1 24123.625,E2 24123.625} C_VEL
LIN {X 0,Y 553.474,Z 504.275,A -85,B 0,C 180,E1 24120.207,E2 24120.207} C_VEL
LIN {X 0,Y 553.5,Z 504.263,A -85,B 0,C 180,E1 24116.893,E2 24116.893} C_VEL
LIN {X 0,Y 553.46,Z 504.288,A -85,B 0,C 180,E1 24113.569,E2 24113.569} C_VEL
LIN {X 0,Y 553.496,Z 504.284,A -85,B 0,C 180,E1 24110.223,E2 24110.223} C_VEL
LIN {X 0,Y 553.477,Z 504.266,A -85,B 0,C 180,E1 24106.949,E2 24106.949} C_VEL
LIN {X 0,Y 553.461,Z 504.27,A -85,B 0,C 180,E1 24103.593,E2 24103.593} C_VEL
LIN {X 0,Y 553.503,Z 504.276,A -85,B 0,C 180,E1 24100.366,E2 24100.366} C_VEL
LIN {X 0,Y 553.456,Z 504.288,A -85,B 0,C 180,E1 24097.124,E2 24097.124} C_VEL
LIN {X 0,Y 553.501,Z 504.282,A -85,B 0,C 180,E1 24093.846,E2 24093.846} C_VEL
LIN {X 0,Y 553.46,Z 504.28,A -85,B 0,C 180,E1 24090.686,E2 24090.686} C_VEL
LIN {X 0,Y 553.465,Z 504.224,A -85,B 0,C 180,E1 24087.304,E2 24087.304} C_VEL
LIN {X 0,Y 553.496,Z 504.285,A -85,B 0,C 180,E1 24084.026,E2 24084.026} C_VEL
LIN {X 0,Y 553.445,Z 504.228,A -85,B 0,C 180,E1 24080.777,E2 24080.777} C_VEL
LIN {X 0,Y 553.535,Z 504.707,A -85,B 0,C 180,E1 24080.199,E2 24080.199} C_VEL
LIN {X 0,Y 555.292,Z 508.413,A -85,B 0,C 180,E1 24079.591,E2 24079.591} C_VEL
LIN {X 0,Y 562.267,Z 523.344,A -85,B 0,C 180,E1 24077.348,E2 24077.348} C_VEL
LIN {X 0,Y 568.846,Z 537.868,A -85,B 0,C 180,E1 24075.323,E2 24075.323} C_VEL
LIN {X 0,Y 571.896,Z 544.714,A -85,B 0,C 180,E1 24074.457,E2 24074.457} C_VEL
LIN {X 0,Y 585.898,Z 567.045,A -85,B 0,C 180,E1 24072.899,E2 24072.899} C_VEL
LIN {X 0,Y 588.995,Z 572.604,A -85,B 0,C 180,E1 24072.56,E2 24072.56} C_VEL
LIN {X 0,Y 582.476,Z 815.584,A -85,B 0,C 180,E1 24069.102,E2 24069.102} C_VEL
LIN {X 0,Y 579.681,Z 921.781,A -85,B 0,C 180,E1 24067.57,E2 24067.57} C_VEL
LIN {X 0,Y 578.415,Z 946.609,A -85,B 0,C 180,E1 24067.046,E2 24067.046} C_VEL
LIN {X 0,Y 577.019,Z 967.839,A -85,B 0,C 180,E1 24066.455,E2 24066.455} C_VEL
LIN {X 0,Y 575.099,Z 992.406,A -85,B 0,C 180,E1 24065.586,E2 24065.586} C_VEL
LIN {X 0,Y 573.269,Z 1012.631,A -85,B 0,C 180,E1 24064.712,E2 24064.712} C_VEL
LIN {X 0,Y 570.946,Z 1035.785,A -85,B 0,C 180,E1 24063.528,E2 24063.528} C_VEL
LIN {X 0,Y 568.746,Z 1055.997,A -85,B 0,C 180,E1 24062.305,E2 24062.305} C_VEL
LIN {X 0,Y 566.308,Z 1077.538,A -85,B 0,C 180,E1 24060.798,E2 24060.798} C_VEL
LIN {X 0,Y 564.088,Z 1096.18,A -85,B 0,C 180,E1 24059.289,E2 24059.289} C_VEL
LIN {X 0,Y 561.729,Z 1116.044,A -85,B 0,C 180,E1 24057.452,E2 24057.452} C_VEL
LIN {X 0,Y 559.755,Z 1132.857,A -85,B 0,C 180,E1 24055.668,E2 24055.668} C_VEL
LIN {X 0,Y 557.795,Z 1150.34,A -85,B 0,C 180,E1 24053.561,E2 24053.561} C_VEL
LIN {X 0,Y 556.389,Z 1163.609,A -85,B 0,C 180,E1 24051.727,E2 24051.727} C_VEL
LIN {X 0,Y 555.035,Z 1177.27,A -85,B 0,C 180,E1 24049.577,E2 24049.577} C_VEL
LIN {X 0,Y 553.972,Z 1188.835,A -85,B 0,C 180,E1 24047.434,E2 24047.434} C_VEL
LIN {X 0,Y 553.199,Z 1198.828,A -85,B 0,C 180,E1 24045.3,E2 24045.3} C_VEL
LIN {X 0,Y 552.609,Z 1207.892,A -85,B 0,C 180,E1 24042.965,E2 24042.965} C_VEL
LIN {X 0,Y 552.265,Z 1214.675,A -85,B 0,C 180,E1 24040.853,E2 24040.853} C_VEL
LIN {X 0,Y 552.047,Z 1221.151,A -85,B 0,C 180,E1 24038.331,E2 24038.331} C_VEL
LIN {X 0,Y 551.954,Z 1225.266,A -85,B 0,C 180,E1 24036.135,E2 24036.135} C_VEL
LIN {X 0,Y 551.918,Z 1228.154,A -85,B 0,C 180,E1 24033.947,E2 24033.947} C_VEL
LIN {X 0,Y 551.905,Z 1229.956,A -85,B 0,C 180,E1 24031.35,E2 24031.35} C_VEL
LIN {X 0,Y 551.892,Z 1230.073,A -85,B 0,C 180,E1 24029.17,E2 24029.17} C_VEL
LIN {X 0,Y 551.89,Z 1229.011,A -85,B 0,C 180,E1 24026.988,E2 24026.988} C_VEL
LIN {X 0,Y 551.916,Z 1226.252,A -85,B 0,C 180,E1 24024.49,E2 24024.49} C_VEL
LIN {X 0,Y 551.98,Z 1222.431,A -85,B 0,C 180,E1 24022.297,E2 24022.297} C_VEL
LIN {X 0,Y 552.151,Z 1217.335,A -85,B 0,C 180,E1 24020.094,E2 24020.094} C_VEL
LIN {X 0,Y 552.503,Z 1209.721,A -85,B 0,C 180,E1 24017.564,E2 24017.564} C_VEL
LIN {X 0,Y 552.985,Z 1201.884,A -85,B 0,C 180,E1 24015.444,E2 24015.444} C_VEL
LIN {X 0,Y 553.804,Z 1191.009,A -85,B 0,C 180,E1 24012.994,E2 24012.994} C_VEL
LIN {X 0,Y 554.739,Z 1180.309,A -85,B 0,C 180,E1 24010.96,E2 24010.96} C_VEL
LIN {X 0,Y 556.091,Z 1166.58,A -85,B 0,C 180,E1 24008.703,E2 24008.703} C_VEL
LIN {X 0,Y 557.53,Z 1152.798,A -85,B 0,C 180,E1 24006.763,E2 24006.763} C_VEL
LIN {X 0,Y 559.377,Z 1136.272,A -85,B 0,C 180,E1 24004.71,E2 24004.71} C_VEL
LIN {X 0,Y 561.442,Z 1118.525,A -85,B 0,C 180,E1 24002.801,E2 24002.801} C_VEL
LIN {X 0,Y 563.716,Z 1099.344,A -85,B 0,C 180,E1 24000.981,E2 24000.981} C_VEL
LIN {X 0,Y 565.866,Z 1081.094,A -85,B 0,C 180,E1 23999.479,E2 23999.479} C_VEL
LIN {X 0,Y 568.319,Z 1060.164,A -85,B 0,C 180,E1 23997.965,E2 23997.965} C_VEL
LIN {X 0,Y 570.561,Z 1039.295,A -85,B 0,C 180,E1 23996.676,E2 23996.676} C_VEL
LIN {X 0,Y 572.9,Z 1016.485,A -85,B 0,C 180,E1 23995.466,E2 23995.466} C_VEL
LIN {X 0,Y 574.871,Z 994.868,A -85,B 0,C 180,E1 23994.516,E2 23994.516} C_VEL
LIN {X 0,Y 576.787,Z 971.302,A -85,B 0,C 180,E1 23993.653,E2 23993.653} C_VEL
LIN {X 0,Y 578.282,Z 948.695,A -85,B 0,C 180,E1 23993.009,E2 23993.009} C_VEL
LIN {X 0,Y 579.529,Z 925.839,A -85,B 0,C 180,E1 23992.503,E2 23992.503} C_VEL
LIN {X 0,Y 580.756,Z 884.065,A -85,B 0,C 180,E1 23991.874,E2 23991.874} C_VEL
LIN {X 0,Y 587.077,Z 641.941,A -85,B 0,C 180,E1 23988.421,E2 23988.421} C_VEL
LIN {X 0,Y 588.838,Z 571.957,A -85,B 0,C 180,E1 23987.42,E2 23987.42} C_VEL
LIN {X 0,Y 574.227,Z 548.378,A -85,B 0,C 180,E1 23985.823,E2 23985.823} C_VEL
LIN {X 0,Y 571.49,Z 543.948,A -85,B 0,C 180,E1 23985.477,E2 23985.477} C_VEL
LIN {X 0,Y 563.314,Z 525.388,A -85,B 0,C 180,E1 23982.97,E2 23982.97} C_VEL
LIN {X 0,Y 557.197,Z 512.538,A -85,B 0,C 180,E1 23981.056,E2 23981.056} C_VEL
LIN {X 0,Y 553.527,Z 504.646,A -85,B 0,C 180,E1 23979.802,E2 23979.802} C_VEL
LIN {X 0,Y 553.457,Z 504.226,A -85,B 0,C 180,E1 23978.955,E2 23978.955} C_VEL
LIN {X 0,Y 553.463,Z 504.271,A -85,B 0,C 180,E1 23975.572,E2 23975.572} C_VEL
LIN {X 0,Y 553.497,Z 504.227,A -85,B 0,C 180,E1 23972.284,E2 23972.284} C_VEL
LIN {X 0,Y 553.456,Z 504.277,A -85,B 0,C 180,E1 23969.077,E2 23969.077} C_VEL
LIN {X 0,Y 553.503,Z 504.274,A -85,B 0,C 180,E1 23965.808,E2 23965.808} C_VEL
LIN {X 0,Y 553.466,Z 504.286,A -85,B 0,C 180,E1 23962.52,E2 23962.52} C_VEL
LIN {X 0,Y 553.471,Z 504.289,A -85,B 0,C 180,E1 23959.086,E2 23959.086} C_VEL
LIN {X 0,Y 553.502,Z 504.272,A -85,B 0,C 180,E1 23955.83,E2 23955.83} C_VEL
LIN {X 0,Y 553.458,Z 504.266,A -85,B 0,C 180,E1 23952.521,E2 23952.521} C_VEL
LIN {X 0,Y 553.5,Z 504.271,A -85,B 0,C 180,E1 23949.252,E2 23949.252} C_VEL
LIN {X 0,Y 553.473,Z 504.283,A -85,B 0,C 180,E1 23946.015,E2 23946.015} C_VEL
LIN {X 0,Y 553.471,Z 504.272,A -85,B 0,C 180,E1 23942.558,E2 23942.558} C_VEL
LIN {X 0,Y 553.503,Z 504.264,A -85,B 0,C 180,E1 23939.275,E2 23939.275} C_VEL
LIN {X 0,Y 553.466,Z 504.284,A -85,B 0,C 180,E1 23935.96,E2 23935.96} C_VEL
LIN {X 0,Y 553.503,Z 504.277,A -85,B 0,C 180,E1 23932.622,E2 23932.622} C_VEL
LIN {X 0,Y 553.492,Z 504.261,A -85,B 0,C 180,E1 23929.276,E2 23929.276} C_VEL
LIN {X 0,Y 553.468,Z 504.269,A -85,B 0,C 180,E1 23925.884,E2 23925.884} C_VEL
LIN {X 0,Y 553.504,Z 504.283,A -85,B 0,C 180,E1 23922.55,E2 23922.55} C_VEL
LIN {X 0,Y 553.486,Z 504.284,A -85,B 0,C 180,E1 23919.152,E2 23919.152} C_VEL
LIN {X 0,Y 553.482,Z 504.28,A -85,B 0,C 180,E1 23915.79,E2 23915.79} C_VEL
LIN {X 0,Y 553.503,Z 504.272,A -85,B 0,C 180,E1 23912.454,E2 23912.454} C_VEL
LIN {X 0,Y 553.475,Z 504.276,A -85,B 0,C 180,E1 23909.132,E2 23909.132} C_VEL
LIN {X 0,Y 553.498,Z 504.274,A -85,B 0,C 180,E1 23905.818,E2 23905.818} C_VEL
LIN {X 0,Y 553.493,Z 504.222,A -85,B 0,C 180,E1 23902.47,E2 23902.47} C_VEL
LIN {X 0,Y 553.536,Z 504.521,A -85,B 0,C 180,E1 23899.776,E2 23899.776} C_VEL
LIN {X 0,Y 555.084,Z 508.192,A -85,B 0,C 180,E1 23899.159,E2 23899.159} C_VEL
LIN {X 0,Y 561.594,Z 522.087,A -85,B 0,C 180,E1 23897.006,E2 23897.006} C_VEL
LIN {X 0,Y 569.454,Z 539.988,A -85,B 0,C 180,E1 23894.473,E2 23894.473} C_VEL
LIN {X 0,Y 577.025,Z 558.819,A -85,B 0,C 180,E1 23892.053,E2 23892.053} C_VEL
LIN {X 0,Y 580.456,Z 568.746,A -85,B 0,C 180,E1 23890.886,E2 23890.886} C_VEL
LIN {X 0,Y 576.195,Z 612.057,A -85,B 0,C 180,E1 23887.586,E2 23887.586} C_VEL
LIN {X 0,Y 574.116,Z 636.355,A -85,B 0,C 180,E1 23885.795,E2 23885.795} C_VEL
LIN {X 0,Y 582.72,Z 685.793,A -85,B 0,C 180,E1 23884.392,E2 23884.392} C_VEL
LIN {X 0,Y 580.725,Z 804.58,A -85,B 0,C 180,E1 23882.904,E2 23882.904} C_VEL
LIN {X 0,Y 579.815,Z 812.282,A -85,B 0,C 180,E1 23882.866,E2 23882.866} C_VEL
LIN {X 0,Y 574.461,Z 832.816,A -85,B 0,C 180,E1 23882.98,E2 23882.98} C_VEL
LIN {X 0,Y 573.745,Z 839.427,A -85,B 0,C 180,E1 23882.942,E2 23882.942} C_VEL
LIN {X 0,Y 571.785,Z 954.278,A -85,B 0,C 180,E1 23881.492,E2 23881.492} C_VEL
LIN {X 0,Y 570.632,Z 976.103,A -85,B 0,C 180,E1 23881.058,E2 23881.058} C_VEL
LIN {X 0,Y 569.105,Z 997.616,A -85,B 0,C 180,E1 23880.455,E2 23880.455} C_VEL
LIN {X 0,Y 567.327,Z 1017.146,A -85,B 0,C 180,E1 23879.736,E2 23879.736} C_VEL
LIN {X 0,Y 565.04,Z 1038.115,A -85,B 0,C 180,E1 23878.771,E2 23878.771} C_VEL
LIN {X 0,Y 562.682,Z 1057.434,A -85,B 0,C 180,E1 23877.689,E2 23877.689} C_VEL
LIN {X 0,Y 560.183,Z 1075.53,A -85,B 0,C 180,E1 23876.461,E2 23876.461} C_VEL
LIN {X 0,Y 557.385,Z 1094.573,A -85,B 0,C 180,E1 23874.933,E2 23874.933} C_VEL
LIN {X 0,Y 554.873,Z 1111.238,A -85,B 0,C 180,E1 23873.355,E2 23873.355} C_VEL
LIN {X 0,Y 552.5,Z 1126.342,A -85,B 0,C 180,E1 23871.665,E2 23871.665} C_VEL
LIN {X 0,Y 550.25,Z 1141.125,A -85,B 0,C 180,E1 23869.73,E2 23869.73} C_VEL
LIN {X 0,Y 548.47,Z 1153.536,A -85,B 0,C 180,E1 23867.834,E2 23867.834} C_VEL
LIN {X 0,Y 546.895,Z 1165.223,A -85,B 0,C 180,E1 23865.699,E2 23865.699} C_VEL
LIN {X 0,Y 545.697,Z 1175.481,A -85,B 0,C 180,E1 23863.456,E2 23863.456} C_VEL
LIN {X 0,Y 544.891,Z 1183.919,A -85,B 0,C 180,E1 23861.216,E2 23861.216} C_VEL
LIN {X 0,Y 544.388,Z 1190.542,A -85,B 0,C 180,E1 23858.982,E2 23858.982} C_VEL
LIN {X 0,Y 544.09,Z 1196.033,A -85,B 0,C 180,E1 23856.542,E2 23856.542} C_VEL
LIN {X 0,Y 543.982,Z 1199.683,A -85,B 0,C 180,E1 23854.216,E2 23854.216} C_VEL
LIN {X 0,Y 543.941,Z 1201.657,A -85,B 0,C 180,E1 23851.896,E2 23851.896} C_VEL
LIN {X 0,Y 543.924,Z 1202.155,A -85,B 0,C 180,E1 23849.473,E2 23849.473} C_VEL
LIN {X 0,Y 543.947,Z 1201.136,A -85,B 0,C 180,E1 23847.155,E2 23847.155} C_VEL
LIN {X 0,Y 544.001,Z 1198.479,A -85,B 0,C 180,E1 23844.833,E2 23844.833} C_VEL
LIN {X 0,Y 544.182,Z 1194.08,A -85,B 0,C 180,E1 23842.398,E2 23842.398} C_VEL
LIN {X 0,Y 544.528,Z 1188.487,A -85,B 0,C 180,E1 23840.168,E2 23840.168} C_VEL
LIN {X 0,Y 545.119,Z 1181.205,A -85,B 0,C 180,E1 23837.93,E2 23837.93} C_VEL
LIN {X 0,Y 546.063,Z 1172.235,A -85,B 0,C 180,E1 23835.689,E2 23835.689} C_VEL
LIN {X 0,Y 547.336,Z 1161.843,A -85,B 0,C 180,E1 23833.552,E2 23833.552} C_VEL
LIN {X 0,Y 548.939,Z 1150.069,A -85,B 0,C 180,E1 23831.523,E2 23831.523} C_VEL
LIN {X 0,Y 550.885,Z 1137.061,A -85,B 0,C 180,E1 23829.606,E2 23829.606} C_VEL
LIN {X 0,Y 553.095,Z 1122.614,A -85,B 0,C 180,E1 23827.801,E2 23827.801} C_VEL
LIN {X 0,Y 555.535,Z 1106.791,A -85,B 0,C 180,E1 23826.112,E2 23826.112} C_VEL
LIN {X 0,Y 558.091,Z 1090.199,A -85,B 0,C 180,E1 23824.591,E2 23824.591} C_VEL
LIN {X 0,Y 560.646,Z 1072.37,A -85,B 0,C 180,E1 23823.217,E2 23823.217} C_VEL
LIN {X 0,Y 563.269,Z 1052.722,A -85,B 0,C 180,E1 23821.94,E2 23821.94} C_VEL
LIN {X 0,Y 565.598,Z 1033.776,A -85,B 0,C 180,E1 23820.913,E2 23820.913} C_VEL
LIN {X 0,Y 567.655,Z 1013.944,A -85,B 0,C 180,E1 23820.043,E2 23820.043} C_VEL
LIN {X 0,Y 569.504,Z 992.634,A -85,B 0,C 180,E1 23819.295,E2 23819.295} C_VEL
LIN {X 0,Y 570.929,Z 971.835,A -85,B 0,C 180,E1 23818.748,E2 23818.748} C_VEL
LIN {X 0,Y 571.95,Z 949.581,A -85,B 0,C 180,E1 23818.347,E2 23818.347} C_VEL
LIN {X 0,Y 576.386,Z 686.777,A -85,B 0,C 180,E1 23815.03,E2 23815.03} C_VEL
LIN {X 0,Y 567.576,Z 635.921,A -85,B 0,C 180,E1 23813.556,E2 23813.556} C_VEL
LIN {X 0,Y 567.569,Z 633.075,A -85,B 0,C 180,E1 23813.393,E2 23813.393} C_VEL
LIN {X 0,Y 571.946,Z 588.947,A -85,B 0,C 180,E1 23810.025,E2 23810.025} C_VEL
LIN {X 0,Y 573.682,Z 571.463,A -85,B 0,C 180,E1 23808.658,E2 23808.658} C_VEL
LIN {X 0,Y 565.964,Z 551.247,A -85,B 0,C 180,E1 23806.122,E2 23806.122} C_VEL
LIN {X 0,Y 558.259,Z 533.021,A -85,B 0,C 180,E1 23803.596,E2 23803.596} C_VEL
LIN {X 0,Y 551.055,Z 517.344,A -85,B 0,C 180,E1 23801.198,E2 23801.198} C_VEL
LIN {X 0,Y 546.903,Z 508.786,A -85,B 0,C 180,E1 23799.784,E2 23799.784} C_VEL
LIN {X 0,Y 545.556,Z 505.409,A -85,B 0,C 180,E1 23799.173,E2 23799.173} C_VEL
LIN {X 0,Y 545.56,Z 505.239,A -85,B 0,C 180,E1 23796.038,E2 23796.038} C_VEL
LIN {X 0,Y 545.531,Z 505.266,A -85,B 0,C 180,E1 23792.727,E2 23792.727} C_VEL
LIN {X 0,Y 545.567,Z 505.263,A -85,B 0,C 180,E1 23789.418,E2 23789.418} C_VEL
LIN {X 0,Y 545.547,Z 505.259,A -85,B 0,C 180,E1 23786.096,E2 23786.096} C_VEL
LIN {X 0,Y 545.529,Z 505.255,A -85,B 0,C 180,E1 23782.638,E2 23782.638} C_VEL
LIN {X 0,Y 545.564,Z 505.251,A -85,B 0,C 180,E1 23779.374,E2 23779.374} C_VEL
LIN {X 0,Y 545.531,Z 505.27,A -85,B 0,C 180,E1 23776.067,E2 23776.067} C_VEL
LIN {X 0,Y 545.541,Z 505.274,A -85,B 0,C 180,E1 23772.598,E2 23772.598} C_VEL
LIN {X 0,Y 545.561,Z 505.258,A -85,B 0,C 180,E1 23769.281,E2 23769.281} C_VEL
LIN {X 0,Y 545.522,Z 505.255,A -85,B 0,C 180,E1 23765.997,E2 23765.997} C_VEL
LIN {X 0,Y 545.56,Z 505.265,A -85,B 0,C 180,E1 23762.626,E2 23762.626} C_VEL
LIN {X 0,Y 545.547,Z 505.272,A -85,B 0,C 180,E1 23759.265,E2 23759.265} C_VEL
LIN {X 0,Y 545.522,Z 505.257,A -85,B 0,C 180,E1 23755.901,E2 23755.901} C_VEL
LIN {X 0,Y 545.567,Z 505.251,A -85,B 0,C 180,E1 23752.629,E2 23752.629} C_VEL
LIN {X 0,Y 545.523,Z 505.278,A -85,B 0,C 180,E1 23749.332,E2 23749.332} C_VEL
LIN {X 0,Y 545.54,Z 505.273,A -85,B 0,C 180,E1 23745.891,E2 23745.891} C_VEL
LIN {X 0,Y 545.552,Z 505.254,A -85,B 0,C 180,E1 23742.618,E2 23742.618} C_VEL
LIN {X 0,Y 545.517,Z 505.258,A -85,B 0,C 180,E1 23739.283,E2 23739.283} C_VEL
LIN {X 0,Y 545.566,Z 505.258,A -85,B 0,C 180,E1 23735.991,E2 23735.991} C_VEL
LIN {X 0,Y 545.524,Z 505.273,A -85,B 0,C 180,E1 23732.727,E2 23732.727} C_VEL
LIN {X 0,Y 545.527,Z 505.27,A -85,B 0,C 180,E1 23729.244,E2 23729.244} C_VEL
LIN {X 0,Y 545.557,Z 505.207,A -85,B 0,C 180,E1 23725.934,E2 23725.934} C_VEL
LIN {X 0,Y 545.51,Z 505.245,A -85,B 0,C 180,E1 23722.7,E2 23722.7} C_VEL
LIN {X 0,Y 545.565,Z 505.502,A -85,B 0,C 180,E1 23721.145,E2 23721.145} C_VEL
LIN {X 0,Y 546.786,Z 508.67,A -85,B 0,C 180,E1 23720.613,E2 23720.613} C_VEL
LIN {X 0,Y 550.081,Z 515.196,A -85,B 0,C 180,E1 23719.539,E2 23719.539} C_VEL
LIN {X 0,Y 556.083,Z 527.874,A -85,B 0,C 180,E1 23717.601,E2 23717.601} C_VEL
LIN {X 0,Y 563.895,Z 545.244,A -85,B 0,C 180,E1 23715.167,E2 23715.167} C_VEL
LIN {X 0,Y 578.381,Z 568.269,A -85,B 0,C 180,E1 23713.494,E2 23713.494} C_VEL
LIN {X 0,Y 582.708,Z 575.747,A -85,B 0,C 180,E1 23713.013,E2 23713.013} C_VEL
LIN {X 0,Y 575.926,Z 817.676,A -85,B 0,C 180,E1 23709.537,E2 23709.537} C_VEL
LIN {X 0,Y 573.043,Z 922.095,A -85,B 0,C 180,E1 23708.013,E2 23708.013} C_VEL
LIN {X 0,Y 571.72,Z 946.901,A -85,B 0,C 180,E1 23707.484,E2 23707.484} C_VEL
LIN {X 0,Y 570.248,Z 968.379,A -85,B 0,C 180,E1 23706.878,E2 23706.878} C_VEL
LIN {X 0,Y 568.229,Z 992.982,A -85,B 0,C 180,E1 23705.994,E2 23705.994} C_VEL
LIN {X 0,Y 566.368,Z 1012.638,A -85,B 0,C 180,E1 23705.136,E2 23705.136} C_VEL
LIN {X 0,Y 563.963,Z 1035.597,A -85,B 0,C 180,E1 23703.95,E2 23703.95} C_VEL
LIN {X 0,Y 561.639,Z 1055.822,A -85,B 0,C 180,E1 23702.714,E2 23702.714} C_VEL
LIN {X 0,Y 559.068,Z 1077.462,A -85,B 0,C 180,E1 23701.181,E2 23701.181} C_VEL
LIN {X 0,Y 556.817,Z 1095.433,A -85,B 0,C 180,E1 23699.709,E2 23699.709} C_VEL
LIN {X 0,Y 554.447,Z 1114.291,A -85,B 0,C 180,E1 23697.961,E2 23697.961} C_VEL
LIN {X 0,Y 552.28,Z 1131.649,A -85,B 0,C 180,E1 23696.099,E2 23696.099} C_VEL
LIN {X 0,Y 550.228,Z 1148.747,A -85,B 0,C 180,E1 23694.019,E2 23694.019} C_VEL
LIN {X 0,Y 548.639,Z 1162.82,A -85,B 0,C 180,E1 23692.05,E2 23692.05} C_VEL
LIN {X 0,Y 547.204,Z 1176.612,A -85,B 0,C 180,E1 23689.868,E2 23689.868} C_VEL
LIN {X 0,Y 546.093,Z 1188.255,A -85,B 0,C 180,E1 23687.694,E2 23687.694} C_VEL
LIN {X 0,Y 545.312,Z 1197.845,A -85,B 0,C 180,E1 23685.636,E2 23685.636} C_VEL
LIN {X 0,Y 544.655,Z 1207.502,A -85,B 0,C 180,E1 23683.158,E2 23683.158} C_VEL
LIN {X 0,Y 544.281,Z 1214.352,A -85,B 0,C 180,E1 23681.014,E2 23681.014} C_VEL
LIN {X 0,Y 544.06,Z 1220.674,A -85,B 0,C 180,E1 23678.561,E2 23678.561} C_VEL
LIN {X 0,Y 543.958,Z 1225.028,A -85,B 0,C 180,E1 23676.226,E2 23676.226} C_VEL
LIN {X 0,Y 543.921,Z 1227.935,A -85,B 0,C 180,E1 23674.006,E2 23674.006} C_VEL
LIN {X 0,Y 543.906,Z 1229.75,A -85,B 0,C 180,E1 23671.369,E2 23671.369} C_VEL
LIN {X 0,Y 543.892,Z 1229.891,A -85,B 0,C 180,E1 23669.263,E2 23669.263} C_VEL
LIN {X 0,Y 543.891,Z 1228.938,A -85,B 0,C 180,E1 23667.155,E2 23667.155} C_VEL
LIN {X 0,Y 543.908,Z 1226.505,A -85,B 0,C 180,E1 23664.726,E2 23664.726} C_VEL
LIN {X 0,Y 543.974,Z 1222.591,A -85,B 0,C 180,E1 23662.395,E2 23662.395} C_VEL
LIN {X 0,Y 544.142,Z 1217.83,A -85,B 0,C 180,E1 23660.267,E2 23660.267} C_VEL
LIN {X 0,Y 544.487,Z 1210.364,A -85,B 0,C 180,E1 23657.678,E2 23657.678} C_VEL
LIN {X 0,Y 544.987,Z 1202.285,A -85,B 0,C 180,E1 23655.443,E2 23655.443} C_VEL
LIN {X 0,Y 545.784,Z 1192.057,A -85,B 0,C 180,E1 23653.065,E2 23653.065} C_VEL
LIN {X 0,Y 546.844,Z 1180.257,A -85,B 0,C 180,E1 23650.785,E2 23650.785} C_VEL
LIN {X 0,Y 548.176,Z 1167.258,A -85,B 0,C 180,E1 23648.605,E2 23648.605} C_VEL
LIN {X 0,Y 549.845,Z 1151.985,A -85,B 0,C 180,E1 23646.418,E2 23646.418} C_VEL
LIN {X 0,Y 551.818,Z 1135.514,A -85,B 0,C 180,E1 23644.339,E2 23644.339} C_VEL
LIN {X 0,Y 553.916,Z 1118.512,A -85,B 0,C 180,E1 23642.477,E2 23642.477} C_VEL
LIN {X 0,Y 556.28,Z 1099.754,A -85,B 0,C 180,E1 23640.665,E2 23640.665} C_VEL
LIN {X 0,Y 558.622,Z 1080.895,A -85,B 0,C 180,E1 23639.09,E2 23639.09} C_VEL
LIN {X 0,Y 561.176,Z 1060.107,A -85,B 0,C 180,E1 23637.568,E2 23637.568} C_VEL
LIN {X 0,Y 563.528,Z 1039.264,A -85,B 0,C 180,E1 23636.265,E2 23636.265} C_VEL
LIN {X 0,Y 565.949,Z 1016.852,A -85,B 0,C 180,E1 23635.062,E2 23635.062} C_VEL
LIN {X 0,Y 567.982,Z 995.536,A -85,B 0,C 180,E1 23634.112,E2 23634.112} C_VEL
LIN {X 0,Y 569.944,Z 972.674,A -85,B 0,C 180,E1 23633.258,E2 23633.258} C_VEL
LIN {X 0,Y 571.57,Z 949.185,A -85,B 0,C 180,E1 23632.577,E2 23632.577} C_VEL
LIN {X 0,Y 572.834,Z 926.965,A -85,B 0,C 180,E1 23632.079,E2 23632.079} C_VEL
LIN {X 0,Y 574.023,Z 889.868,A -85,B 0,C 180,E1 23631.504,E2 23631.504} C_VEL
LIN {X 0,Y 580.663,Z 646.541,A -85,B 0,C 180,E1 23627.998,E2 23627.998} C_VEL
LIN {X 0,Y 582.555,Z 575.148,A -85,B 0,C 180,E1 23626.968,E2 23626.968} C_VEL
LIN {X 0,Y 568.302,Z 552.19,A -85,B 0,C 180,E1 23625.373,E2 23625.373} C_VEL
LIN {X 0,Y 563.815,Z 545.078,A -85,B 0,C 180,E1 23624.818,E2 23624.818} C_VEL
LIN {X 0,Y 556.532,Z 528.879,A -85,B 0,C 180,E1 23622.558,E2 23622.558} C_VEL
LIN {X 0,Y 551.012,Z 517.219,A -85,B 0,C 180,E1 23620.789,E2 23620.789} C_VEL
LIN {X 0,Y 547.117,Z 509.141,A -85,B 0,C 180,E1 23619.494,E2 23619.494} C_VEL
LIN {X 0,Y 545.567,Z 505.522,A -85,B 0,C 180,E1 23618.882,E2 23618.882} C_VEL
LIN {X 0,Y 545.513,Z 505.238,A -85,B 0,C 180,E1 23617.474,E2 23617.474} C_VEL
LIN {X 0,Y 545.558,Z 505.21,A -85,B 0,C 180,E1 23614.241,E2 23614.241} C_VEL
LIN {X 0,Y 545.519,Z 505.263,A -85,B 0,C 180,E1 23610.932,E2 23610.932} C_VEL
LIN {X 0,Y 545.551,Z 505.263,A -85,B 0,C 180,E1 23607.626,E2 23607.626} C_VEL
LIN {X 0,Y 545.543,Z 505.257,A -85,B 0,C 180,E1 23604.355,E2 23604.355} C_VEL
LIN {X 0,Y 545.525,Z 505.257,A -85,B 0,C 180,E1 23601.054,E2 23601.054} C_VEL
LIN {X 0,Y 545.565,Z 505.26,A -85,B 0,C 180,E1 23597.823,E2 23597.823} C_VEL
LIN {X 0,Y 545.522,Z 505.276,A -85,B 0,C 180,E1 23594.543,E2 23594.543} C_VEL
LIN {X 0,Y 545.557,Z 505.264,A -85,B 0,C 180,E1 23591.202,E2 23591.202} C_VEL
LIN {X 0,Y 545.542,Z 505.247,A -85,B 0,C 180,E1 23587.901,E2 23587.901} C_VEL
LIN {X 0,Y 545.527,Z 505.26,A -85,B 0,C 180,E1 23584.52,E2 23584.52} C_VEL
LIN {X 0,Y 545.566,Z 505.273,A -85,B 0,C 180,E1 23581.155,E2 23581.155} C_VEL
LIN {X 0,Y 545.529,Z 505.263,A -85,B 0,C 180,E1 23577.899,E2 23577.899} C_VEL
LIN {X 0,Y 545.547,Z 505.253,A -85,B 0,C 180,E1 23574.531,E2 23574.531} C_VEL
LIN {X 0,Y 545.564,Z 505.271,A -85,B 0,C 180,E1 23571.144,E2 23571.144} C_VEL
LIN {X 0,Y 545.531,Z 505.277,A -85,B 0,C 180,E1 23567.832,E2 23567.832} C_VEL
LIN {X 0,Y 545.562,Z 505.254,A -85,B 0,C 180,E1 23564.479,E2 23564.479} C_VEL
LIN {X 0,Y 545.552,Z 505.252,A -85,B 0,C 180,E1 23561.07,E2 23561.07} C_VEL
LIN {X 0,Y 545.535,Z 505.26,A -85,B 0,C 180,E1 23557.703,E2 23557.703} C_VEL
LIN {X 0,Y 545.562,Z 505.267,A -85,B 0,C 180,E1 23554.371,E2 23554.371} C_VEL
LIN {X 0,Y 545.541,Z 505.275,A -85,B 0,C 180,E1 23551.061,E2 23551.061} C_VEL
LIN {X 0,Y 545.551,Z 505.271,A -85,B 0,C 180,E1 23547.644,E2 23547.644} C_VEL
LIN {X 0,Y 545.558,Z 505.253,A -85,B 0,C 180,E1 23544.221,E2 23544.221} C_VEL
LIN {X 0,Y 545.539,Z 505.268,A -85,B 0,C 180,E1 23540.913,E2 23540.913} C_VEL
LIN {X 0,Y 545.635,Z 505.781,A -85,B 0,C 180,E1 23540.61,E2 23540.61} C_VEL
LIN {X 0,Y 547.343,Z 509.423,A -85,B 0,C 180,E1 23539.981,E2 23539.981} C_VEL
LIN {X 0,Y 553.867,Z 523.407,A -85,B 0,C 180,E1 23537.744,E2 23537.744} C_VEL
LIN {X 0,Y 560.999,Z 539.371,A -85,B 0,C 180,E1 23535.393,E2 23535.393} C_VEL
LIN {X 0,Y 568.656,Z 558.22,A -85,B 0,C 180,E1 23532.879,E2 23532.879} C_VEL
LIN {X 0,Y 573.731,Z 571.842,A -85,B 0,C 180,E1 23531.205,E2 23531.205} C_VEL
LIN {X 0,Y 569.264,Z 615.162,A -85,B 0,C 180,E1 23527.869,E2 23527.869} C_VEL
LIN {X 0,Y 567.465,Z 635.476,A -85,B 0,C 180,E1 23526.36,E2 23526.36} C_VEL
LIN {X 0,Y 576.385,Z 687.058,A -85,B 0,C 180,E1 23524.866,E2 23524.866} C_VEL
LIN {X 0,Y 573.745,Z 839.427,A -85,B 0,C 180,E1 23522.942,E2 23522.942} C_VEL
LIN {X 0,Y 572.811,Z 847.13,A -85,B 0,C 180,E1 23522.906,E2 23522.906} C_VEL
LIN {X 0,Y 567.43,Z 867.656,A -85,B 0,C 180,E1 23523.023,E2 23523.023} C_VEL
LIN {X 0,Y 566.724,Z 874.265,A -85,B 0,C 180,E1 23522.984,E2 23522.984} C_VEL
LIN {X 0,Y 565.218,Z 954.826,A -85,B 0,C 180,E1 23521.95,E2 23521.95} C_VEL
LIN {X 0,Y 563.99,Z 976.648,A -85,B 0,C 180,E1 23521.505,E2 23521.505} C_VEL
LIN {X 0,Y 562.318,Z 998.796,A -85,B 0,C 180,E1 23520.869,E2 23520.869} C_VEL
LIN {X 0,Y 560.442,Z 1018.483,A -85,B 0,C 180,E1 23520.129,E2 23520.129} C_VEL
LIN {X 0,Y 558.08,Z 1038.988,A -85,B 0,C 180,E1 23519.164,E2 23519.164} C_VEL
LIN {X 0,Y 555.622,Z 1058.136,A -85,B 0,C 180,E1 23518.072,E2 23518.072} C_VEL
LIN {X 0,Y 553.023,Z 1076.192,A -85,B 0,C 180,E1 23516.829,E2 23516.829} C_VEL
LIN {X 0,Y 550.201,Z 1094.519,A -85,B 0,C 180,E1 23515.338,E2 23515.338} C_VEL
LIN {X 0,Y 547.566,Z 1111.208,A -85,B 0,C 180,E1 23513.743,E2 23513.743} C_VEL
LIN {X 0,Y 544.999,Z 1126.776,A -85,B 0,C 180,E1 23511.978,E2 23511.978} C_VEL
LIN {X 0,Y 542.663,Z 1141.349,A -85,B 0,C 180,E1 23510.042,E2 23510.042} C_VEL
LIN {X 0,Y 540.762,Z 1153.887,A -85,B 0,C 180,E1 23508.097,E2 23508.097} C_VEL
LIN {X 0,Y 539.096,Z 1165.547,A -85,B 0,C 180,E1 23505.932,E2 23505.932} C_VEL
LIN {X 0,Y 537.824,Z 1175.773,A -85,B 0,C 180,E1 23503.657,E2 23503.657} C_VEL
LIN {X 0,Y 536.969,Z 1184.183,A -85,B 0,C 180,E1 23501.384,E2 23501.384} C_VEL
LIN {X 0,Y 536.428,Z 1190.792,A -85,B 0,C 180,E1 23499.116,E2 23499.116} C_VEL
LIN {X 0,Y 536.106,Z 1196.262,A -85,B 0,C 180,E1 23496.64,E2 23496.64} C_VEL
LIN {X 0,Y 535.988,Z 1199.897,A -85,B 0,C 180,E1 23494.279,E2 23494.279} C_VEL
LIN {X 0,Y 535.944,Z 1201.864,A -85,B 0,C 180,E1 23491.924,E2 23491.924} C_VEL
LIN {X 0,Y 535.928,Z 1202.36,A -85,B 0,C 180,E1 23489.466,E2 23489.466} C_VEL
LIN {X 0,Y 535.951,Z 1201.344,A -85,B 0,C 180,E1 23487.113,E2 23487.113} C_VEL
LIN {X 0,Y 536.012,Z 1198.698,A -85,B 0,C 180,E1 23484.756,E2 23484.756} C_VEL
LIN {X 0,Y 536.205,Z 1194.316,A -85,B 0,C 180,E1 23482.284,E2 23482.284} C_VEL
LIN {X 0,Y 536.578,Z 1188.737,A -85,B 0,C 180,E1 23480.021,E2 23480.021} C_VEL
LIN {X 0,Y 537.222,Z 1181.398,A -85,B 0,C 180,E1 23477.728,E2 23477.728} C_VEL
LIN {X 0,Y 538.238,Z 1172.364,A -85,B 0,C 180,E1 23475.437,E2 23475.437} C_VEL
LIN {X 0,Y 539.568,Z 1162.162,A -85,B 0,C 180,E1 23473.308,E2 23473.308} C_VEL
LIN {X 0,Y 541.258,Z 1150.424,A -85,B 0,C 180,E1 23471.251,E2 23471.251} C_VEL
LIN {X 0,Y 543.303,Z 1137.464,A -85,B 0,C 180,E1 23469.308,E2 23469.308} C_VEL
LIN {X 0,Y 545.625,Z 1123.039,A -85,B 0,C 180,E1 23467.481,E2 23467.481} C_VEL
LIN {X 0,Y 548.261,Z 1106.743,A -85,B 0,C 180,E1 23465.717,E2 23465.717} C_VEL
LIN {X 0,Y 550.946,Z 1090.125,A -85,B 0,C 180,E1 23464.18,E2 23464.18} C_VEL
LIN {X 0,Y 553.578,Z 1072.528,A -85,B 0,C 180,E1 23462.809,E2 23462.809} C_VEL
LIN {X 0,Y 556.356,Z 1052.634,A -85,B 0,C 180,E1 23461.503,E2 23461.503} C_VEL
LIN {X 0,Y 558.79,Z 1033.639,A -85,B 0,C 180,E1 23460.465,E2 23460.465} C_VEL
LIN {X 0,Y 560.93,Z 1013.783,A -85,B 0,C 180,E1 23459.587,E2 23459.587} C_VEL
LIN {X 0,Y 562.871,Z 992.307,A -85,B 0,C 180,E1 23458.829,E2 23458.829} C_VEL
LIN {X 0,Y 564.363,Z 971.469,A -85,B 0,C 180,E1 23458.278,E2 23458.278} C_VEL
LIN {X 0,Y 565.416,Z 949.369,A -85,B 0,C 180,E1 23457.878,E2 23457.878} C_VEL
LIN {X 0,Y 570.101,Z 688.197,A -85,B 0,C 180,E1 23454.548,E2 23454.548} C_VEL
LIN {X 0,Y 561.246,Z 636.592,A -85,B 0,C 180,E1 23453.027,E2 23453.027} C_VEL
LIN {X 0,Y 560.888,Z 633.133,A -85,B 0,C 180,E1 23452.885,E2 23452.885} C_VEL
LIN {X 0,Y 565.401,Z 589.756,A -85,B 0,C 180,E1 23449.534,E2 23449.534} C_VEL
LIN {X 0,Y 567.016,Z 575.195,A -85,B 0,C 180,E1 23448.391,E2 23448.391} C_VEL
LIN {X 0,Y 559.283,Z 554.848,A -85,B 0,C 180,E1 23445.796,E2 23445.796} C_VEL
LIN {X 0,Y 551.664,Z 536.801,A -85,B 0,C 180,E1 23443.246,E2 23443.246} C_VEL
LIN {X 0,Y 545.191,Z 522.587,A -85,B 0,C 180,E1 23441.04,E2 23441.04} C_VEL
LIN {X 0,Y 540.986,Z 513.899,A -85,B 0,C 180,E1 23439.583,E2 23439.583} C_VEL
LIN {X 0,Y 538.876,Z 509.672,A -85,B 0,C 180,E1 23438.841,E2 23438.841} C_VEL
LIN {X 0,Y 537.643,Z 506.382,A -85,B 0,C 180,E1 23438.225,E2 23438.225} C_VEL
LIN {X 0,Y 537.594,Z 506.27,A -85,B 0,C 180,E1 23434.82,E2 23434.82} C_VEL
LIN {X 0,Y 537.626,Z 506.26,A -85,B 0,C 180,E1 23431.383,E2 23431.383} C_VEL
LIN {X 0,Y 537.63,Z 506.256,A -85,B 0,C 180,E1 23427.947,E2 23427.947} C_VEL
LIN {X 0,Y 537.592,Z 506.267,A -85,B 0,C 180,E1 23424.505,E2 23424.505} C_VEL
LIN {X 0,Y 537.627,Z 506.261,A -85,B 0,C 180,E1 23421.15,E2 23421.15} C_VEL
LIN {X 0,Y 537.614,Z 506.252,A -85,B 0,C 180,E1 23417.759,E2 23417.759} C_VEL
LIN {X 0,Y 537.585,Z 506.243,A -85,B 0,C 180,E1 23414.322,E2 23414.322} C_VEL
LIN {X 0,Y 537.623,Z 506.24,A -85,B 0,C 180,E1 23411.044,E2 23411.044} C_VEL
LIN {X 0,Y 537.595,Z 506.267,A -85,B 0,C 180,E1 23407.696,E2 23407.696} C_VEL
LIN {X 0,Y 537.595,Z 506.26,A -85,B 0,C 180,E1 23404.267,E2 23404.267} C_VEL
LIN {X 0,Y 537.625,Z 506.238,A -85,B 0,C 180,E1 23400.959,E2 23400.959} C_VEL
LIN {X 0,Y 537.582,Z 506.256,A -85,B 0,C 180,E1 23397.655,E2 23397.655} C_VEL
LIN {X 0,Y 537.611,Z 506.262,A -85,B 0,C 180,E1 23394.236,E2 23394.236} C_VEL
LIN {X 0,Y 537.612,Z 506.245,A -85,B 0,C 180,E1 23390.904,E2 23390.904} C_VEL
LIN {X 0,Y 537.58,Z 506.243,A -85,B 0,C 180,E1 23387.54,E2 23387.54} C_VEL
LIN {X 0,Y 537.628,Z 506.249,A -85,B 0,C 180,E1 23384.244,E2 23384.244} C_VEL
LIN {X 0,Y 537.592,Z 506.267,A -85,B 0,C 180,E1 23380.877,E2 23380.877} C_VEL
LIN {X 0,Y 537.589,Z 506.264,A -85,B 0,C 180,E1 23377.471,E2 23377.471} C_VEL
LIN {X 0,Y 537.625,Z 506.25,A -85,B 0,C 180,E1 23374.175,E2 23374.175} C_VEL
LIN {X 0,Y 537.578,Z 506.254,A -85,B 0,C 180,E1 23370.835,E2 23370.835} C_VEL
LIN {X 0,Y 537.611,Z 506.198,A -85,B 0,C 180,E1 23367.603,E2 23367.603} C_VEL
LIN {X 0,Y 537.595,Z 506.249,A -85,B 0,C 180,E1 23364.266,E2 23364.266} C_VEL
LIN {X 0,Y 537.639,Z 506.493,A -85,B 0,C 180,E1 23362.093,E2 23362.093} C_VEL
LIN {X 0,Y 539.164,Z 510.031,A -85,B 0,C 180,E1 23361.456,E2 23361.456} C_VEL
LIN {X 0,Y 544.585,Z 521.215,A -85,B 0,C 180,E1 23359.599,E2 23359.599} C_VEL
LIN {X 0,Y 550.564,Z 533.89,A -85,B 0,C 180,E1 23357.64,E2 23357.64} C_VEL
LIN {X 0,Y 556.461,Z 546.88,A -85,B 0,C 180,E1 23355.816,E2 23355.816} C_VEL
LIN {X 0,Y 571.258,Z 570.044,A -85,B 0,C 180,E1 23354.068,E2 23354.068} C_VEL
LIN {X 0,Y 576.457,Z 579.028,A -85,B 0,C 180,E1 23353.474,E2 23353.474} C_VEL
LIN {X 0,Y 569.413,Z 819.659,A -85,B 0,C 180,E1 23349.983,E2 23349.983} C_VEL
LIN {X 0,Y 566.449,Z 922.274,A -85,B 0,C 180,E1 23348.469,E2 23348.469} C_VEL
LIN {X 0,Y 565.069,Z 947.151,A -85,B 0,C 180,E1 23347.934,E2 23347.934} C_VEL
LIN {X 0,Y 563.523,Z 968.837,A -85,B 0,C 180,E1 23347.315,E2 23347.315} C_VEL
LIN {X 0,Y 561.445,Z 993.064,A -85,B 0,C 180,E1 23346.435,E2 23346.435} C_VEL
LIN {X 0,Y 559.514,Z 1012.58,A -85,B 0,C 180,E1 23345.574,E2 23345.574} C_VEL
LIN {X 0,Y 556.996,Z 1035.632,A -85,B 0,C 180,E1 23344.371,E2 23344.371} C_VEL
LIN {X 0,Y 554.541,Z 1055.961,A -85,B 0,C 180,E1 23343.115,E2 23343.115} C_VEL
LIN {X 0,Y 551.861,Z 1077.437,A -85,B 0,C 180,E1 23341.575,E2 23341.575} C_VEL
LIN {X 0,Y 549.418,Z 1096.009,A -85,B 0,C 180,E1 23340.03,E2 23340.03} C_VEL
LIN {X 0,Y 546.784,Z 1115.78,A -85,B 0,C 180,E1 23338.15,E2 23338.15} C_VEL
LIN {X 0,Y 544.663,Z 1132.001,A -85,B 0,C 180,E1 23336.375,E2 23336.375} C_VEL
LIN {X 0,Y 542.507,Z 1148.968,A -85,B 0,C 180,E1 23334.267,E2 23334.267} C_VEL
LIN {X 0,Y 540.831,Z 1162.925,A -85,B 0,C 180,E1 23332.271,E2 23332.271} C_VEL
LIN {X 0,Y 539.323,Z 1176.579,A -85,B 0,C 180,E1 23330.058,E2 23330.058} C_VEL
LIN {X 0,Y 538.17,Z 1188.233,A -85,B 0,C 180,E1 23327.851,E2 23327.851} C_VEL
LIN {X 0,Y 537.285,Z 1198.793,A -85,B 0,C 180,E1 23325.544,E2 23325.544} C_VEL
LIN {X 0,Y 536.649,Z 1207.825,A -85,B 0,C 180,E1 23323.138,E2 23323.138} C_VEL
LIN {X 0,Y 536.286,Z 1214.305,A -85,B 0,C 180,E1 23321.071,E2 23321.071} C_VEL
LIN {X 0,Y 536.061,Z 1220.607,A -85,B 0,C 180,E1 23318.581,E2 23318.581} C_VEL
LIN {X 0,Y 535.958,Z 1224.949,A -85,B 0,C 180,E1 23316.212,E2 23316.212} C_VEL
LIN {X 0,Y 535.921,Z 1227.83,A -85,B 0,C 180,E1 23313.958,E2 23313.958} C_VEL
LIN {X 0,Y 535.912,Z 1229.569,A -85,B 0,C 180,E1 23311.283,E2 23311.283} C_VEL
LIN {X 0,Y 535.898,Z 1229.662,A -85,B 0,C 180,E1 23309.145,E2 23309.145} C_VEL
LIN {X 0,Y 535.895,Z 1228.656,A -85,B 0,C 180,E1 23307.005,E2 23307.005} C_VEL
LIN {X 0,Y 535.922,Z 1225.939,A -85,B 0,C 180,E1 23304.433,E2 23304.433} C_VEL
LIN {X 0,Y 535.989,Z 1222.11,A -85,B 0,C 180,E1 23302.173,E2 23302.173} C_VEL
LIN {X 0,Y 536.163,Z 1216.993,A -85,B 0,C 180,E1 23299.904,E2 23299.904} C_VEL
LIN {X 0,Y 536.553,Z 1209.322,A -85,B 0,C 180,E1 23297.297,E2 23297.297} C_VEL
LIN {X 0,Y 537.098,Z 1201.199,A -85,B 0,C 180,E1 23295.062,E2 23295.062} C_VEL
LIN {X 0,Y 537.979,Z 1190.418,A -85,B 0,C 180,E1 23292.589,E2 23292.589} C_VEL
LIN {X 0,Y 539.015,Z 1179.604,A -85,B 0,C 180,E1 23290.495,E2 23290.495} C_VEL
LIN {X 0,Y 540.506,Z 1165.863,A -85,B 0,C 180,E1 23288.172,E2 23288.172} C_VEL
LIN {X 0,Y 542.198,Z 1151.383,A -85,B 0,C 180,E1 23286.065,E2 23286.065} C_VEL
LIN {X 0,Y 544.329,Z 1134.652,A -85,B 0,C 180,E1 23283.93,E2 23283.93} C_VEL
LIN {X 0,Y 546.471,Z 1118.143,A -85,B 0,C 180,E1 23282.099,E2 23282.099} C_VEL
LIN {X 0,Y 549.008,Z 1099.142,A -85,B 0,C 180,E1 23280.246,E2 23280.246} C_VEL
LIN {X 0,Y 551.405,Z 1080.79,A -85,B 0,C 180,E1 23278.695,E2 23278.695} C_VEL
LIN {X 0,Y 554.039,Z 1060.334,A -85,B 0,C 180,E1 23277.177,E2 23277.177} C_VEL
LIN {X 0,Y 556.524,Z 1039.374,A -85,B 0,C 180,E1 23275.851,E2 23275.851} C_VEL
LIN {X 0,Y 559.037,Z 1017.228,A -85,B 0,C 180,E1 23274.647,E2 23274.647} C_VEL
LIN {X 0,Y 561.202,Z 995.467,A -85,B 0,C 180,E1 23273.667,E2 23273.667} C_VEL
LIN {X 0,Y 563.273,Z 972.227,A -85,B 0,C 180,E1 23272.793,E2 23272.793} C_VEL
LIN {X 0,Y 564.944,Z 948.914,A -85,B 0,C 180,E1 23272.115,E2 23272.115} C_VEL
LIN {X 0,Y 566.323,Z 925.438,A -85,B 0,C 180,E1 23271.588,E2 23271.588} C_VEL
LIN {X 0,Y 567.884,Z 874.629,A -85,B 0,C 180,E1 23270.819,E2 23270.819} C_VEL
LIN {X 0,Y 574.781,Z 634.388,A -85,B 0,C 180,E1 23267.324,E2 23267.324} C_VEL
LIN {X 0,Y 576.304,Z 578.388,A -85,B 0,C 180,E1 23266.507,E2 23266.507} C_VEL
